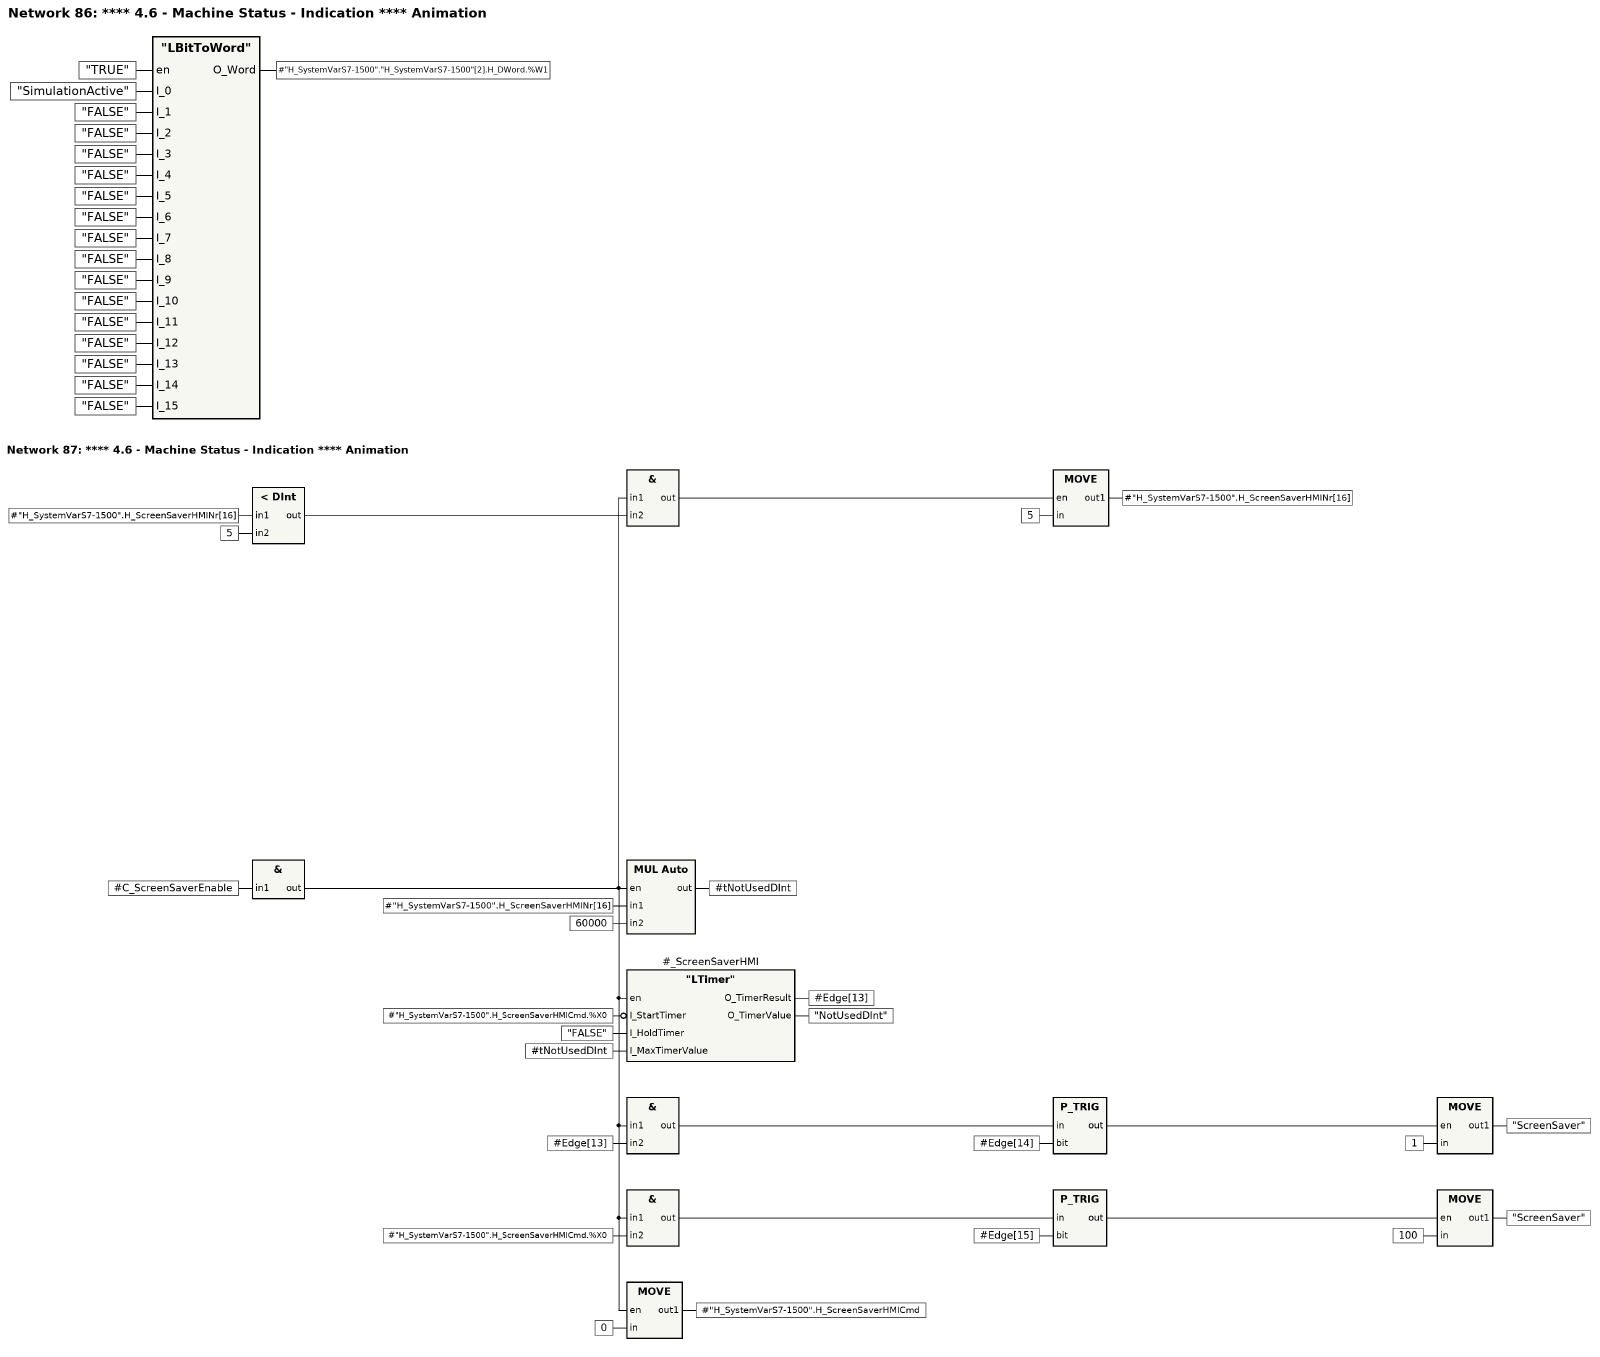
   IF "TRUE" THEN
       "LBitToWord"(I_0 := "SimulationActive",
                    I_1 := "FALSE",
                    I_2 := "FALSE",
                    I_3 := "FALSE",
                    I_4 := "FALSE",
                    I_5 := "FALSE",
                    I_6 := "FALSE",
                    I_7 := "FALSE",
                    I_8 := "FALSE",
                    I_9 := "FALSE",
                    I_10 := "FALSE",
                    I_11 := "FALSE",
                    I_12 := "FALSE",
                    I_13 := "FALSE",
                    I_14 := "FALSE",
                    I_15 := "FALSE",
                    O_Word => #"H_SystemVarS7-1500"."H_SystemVarS7-1500"[2].H_DWord.%W1);
   END_IF;
END_REGION

REGION Network 87: **** 4.6 - Machine Status - Indication **** Animation
   // Animation
   IF #C_ScreenSaverEnable AND (#"H_SystemVarS7-1500".H_ScreenSaverHMINr[16] < 5) THEN
       #"H_SystemVarS7-1500".H_ScreenSaverHMINr[16] := 5;
   END_IF;
   IF #C_ScreenSaverEnable THEN
       #tNotUsedDInt := #"H_SystemVarS7-1500".H_ScreenSaverHMINr[16] * 60000;
       #_ScreenSaverHMI(I_StartTimer := NOT #"H_SystemVarS7-1500".H_ScreenSaverHMICmd.%X0,   // "LTimer"
                        I_HoldTimer := "FALSE",
                        I_MaxTimerValue := #tNotUsedDInt,
                        O_TimerResult => #Edge[13],
                        O_TimerValue => "NotUsedDInt");
   END_IF;
   #_w1 := #C_ScreenSaverEnable AND #Edge[13];
   #_w2 := #_w1 AND NOT #Edge[14];   // rising edge
   #Edge[14] := #_w1;
   IF #_w2 THEN "ScreenSaver" := 1; END_IF;
   #_w3 := #C_ScreenSaverEnable AND #"H_SystemVarS7-1500".H_ScreenSaverHMICmd.%X0;
   #_w4 := #_w3 AND NOT #Edge[15];   // rising edge
   #Edge[15] := #_w3;
   IF #_w4 THEN "ScreenSaver" := 100; END_IF;
   IF #C_ScreenSaverEnable THEN #"H_SystemVarS7-1500".H_ScreenSaverHMICmd := 0; END_IF;
END_REGION

REGION Network 88: **** 4.6 - Machine Status - Indication **** Animation (LED status of the cpu)
   // Animation (LED status of the cpu)
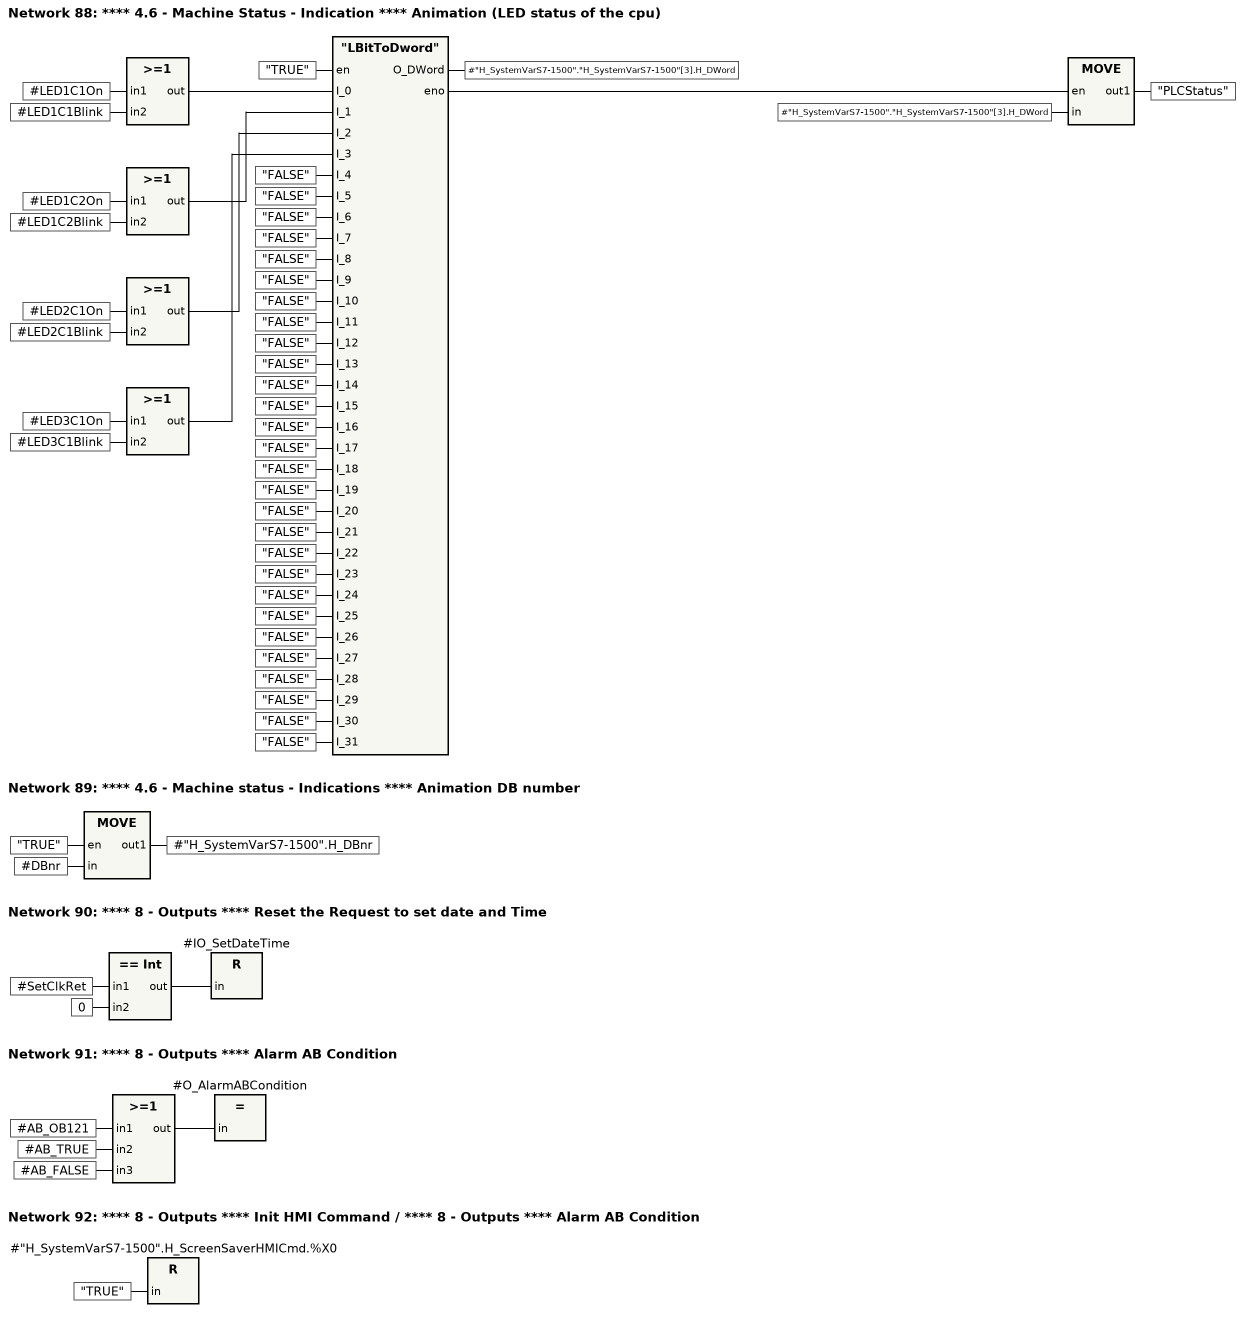
   "LBitToDword"(EN := "TRUE",
                 I_0 := #LED1C1On OR #LED1C1Blink,
                 I_1 := #LED1C2On OR #LED1C2Blink,
                 I_2 := #LED2C1On OR #LED2C1Blink,
                 I_3 := #LED3C1On OR #LED3C1Blink,
                 I_4 := "FALSE",
                 I_5 := "FALSE",
                 I_6 := "FALSE",
                 I_7 := "FALSE",
                 I_8 := "FALSE",
                 I_9 := "FALSE",
                 I_10 := "FALSE",
                 I_11 := "FALSE",
                 I_12 := "FALSE",
                 I_13 := "FALSE",
                 I_14 := "FALSE",
                 I_15 := "FALSE",
                 I_16 := "FALSE",
                 I_17 := "FALSE",
                 I_18 := "FALSE",
                 I_19 := "FALSE",
                 I_20 := "FALSE",
                 I_21 := "FALSE",
                 I_22 := "FALSE",
                 I_23 := "FALSE",
                 I_24 := "FALSE",
                 I_25 := "FALSE",
                 I_26 := "FALSE",
                 I_27 := "FALSE",
                 I_28 := "FALSE",
                 I_29 := "FALSE",
                 I_30 := "FALSE",
                 I_31 := "FALSE",
                 O_DWord => #"H_SystemVarS7-1500"."H_SystemVarS7-1500"[3].H_DWord,
                 ENO => #_w1);
   IF #_w1 THEN "PLCStatus" := #"H_SystemVarS7-1500"."H_SystemVarS7-1500"[3].H_DWord; END_IF;
END_REGION

REGION Network 89: **** 4.6 - Machine status - Indications **** Animation DB number
   // Animation DB number
   IF "TRUE" THEN #"H_SystemVarS7-1500".H_DBnr := #DBnr; END_IF;
END_REGION

REGION Network 90: **** 8 - Outputs **** Reset the Request to set date and Time
   // Reset the Request to set date and Time
   IF #SetClkRet = 0 THEN #IO_SetDateTime := FALSE; END_IF;
END_REGION

REGION Network 91: **** 8 - Outputs **** Alarm AB Condition
   // Alarm AB Condition
   #O_AlarmABCondition := #AB_OB121 OR #AB_TRUE OR #AB_FALSE;
END_REGION

REGION Network 92: **** 8 - Outputs **** Init HMI Command / **** 8 - Outputs **** Alarm AB Condition
   // Init HMI Command / Alarm AB Condition
   IF "TRUE" THEN #"H_SystemVarS7-1500".H_ScreenSaverHMICmd.%X0 := FALSE; END_IF;
END_REGION

REGION Network 93: **** 9 - Alarm Summary **** Alarm A
   // Alarm A
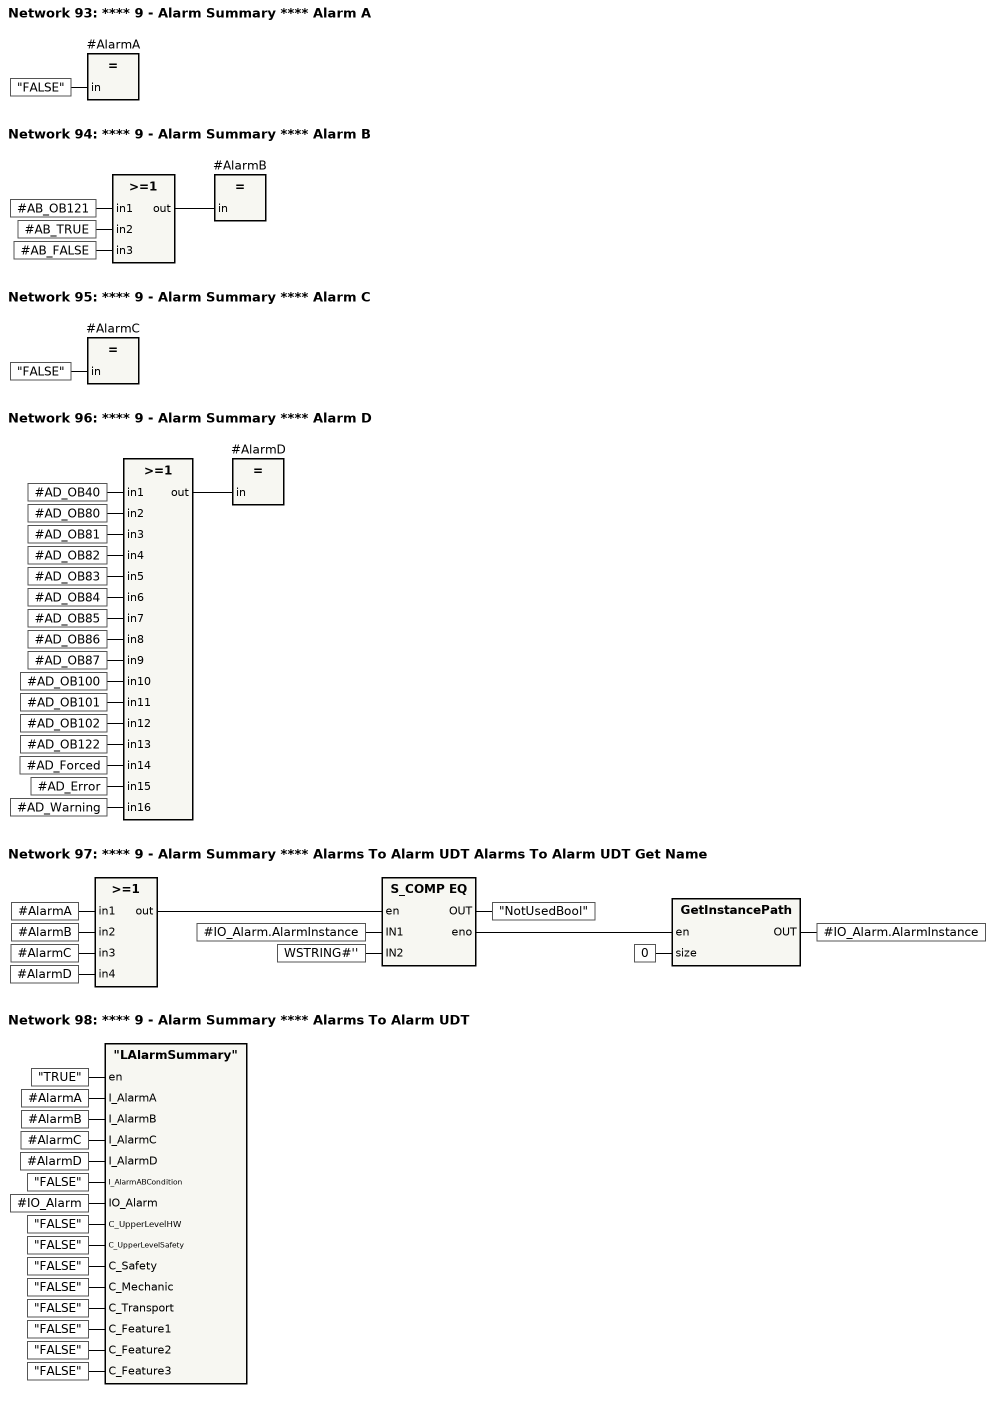
   #AlarmA := "FALSE";
END_REGION

REGION Network 94: **** 9 - Alarm Summary **** Alarm B
   // Alarm B
   #AlarmB := #AB_OB121 OR #AB_TRUE OR #AB_FALSE;
END_REGION

REGION Network 95: **** 9 - Alarm Summary **** Alarm C
   // Alarm C
   #AlarmC := "FALSE";
END_REGION

REGION Network 96: **** 9 - Alarm Summary **** Alarm D
   // Alarm D
   #AlarmD := #AD_OB40 OR #AD_OB80 OR #AD_OB81 OR #AD_OB82 OR #AD_OB83 OR #AD_OB84 OR #AD_OB85 OR #AD_OB86 OR #AD_OB87 OR #AD_OB100 OR #AD_OB101 OR #AD_OB102 OR #AD_OB122 OR #AD_Forced OR #AD_Error OR #AD_Warning;
END_REGION

REGION Network 97: **** 9 - Alarm Summary **** Alarms To Alarm UDT Alarms To Alarm UDT Get Name
   // Alarm / Alarm D
   S_COMP(EN := #AlarmA OR #AlarmB OR #AlarmC OR #AlarmD,
          IN1 := #IO_Alarm.AlarmInstance,
          IN2 := WSTRING#'',
          OUT => "NotUsedBool",
          ENO => #_w1);
   IF #_w1 THEN GetInstancePath(size := 0, OUT => #IO_Alarm.AlarmInstance); END_IF;
END_REGION

REGION Network 98: **** 9 - Alarm Summary **** Alarms To Alarm UDT
   // Alarm / Alarm D
   IF "TRUE" THEN
       "LAlarmSummary"(I_AlarmA := #AlarmA,
                       I_AlarmB := #AlarmB,
                       I_AlarmC := #AlarmC,
                       I_AlarmD := #AlarmD,
                       I_AlarmABCondition := "FALSE",
                       IO_Alarm := #IO_Alarm,
                       C_UpperLevelHW := "FALSE",
                       C_UpperLevelSafety := "FALSE",
                       C_Safety := "FALSE",
                       C_Mechanic := "FALSE",
                       C_Transport := "FALSE",
                       C_Feature1 := "FALSE",
                       C_Feature2 := "FALSE",
                       C_Feature3 := "FALSE");
   END_IF;
END_REGION

REGION Network 99: **** 9.1 - Alarm Output **** Alarm A
   // Alarm A
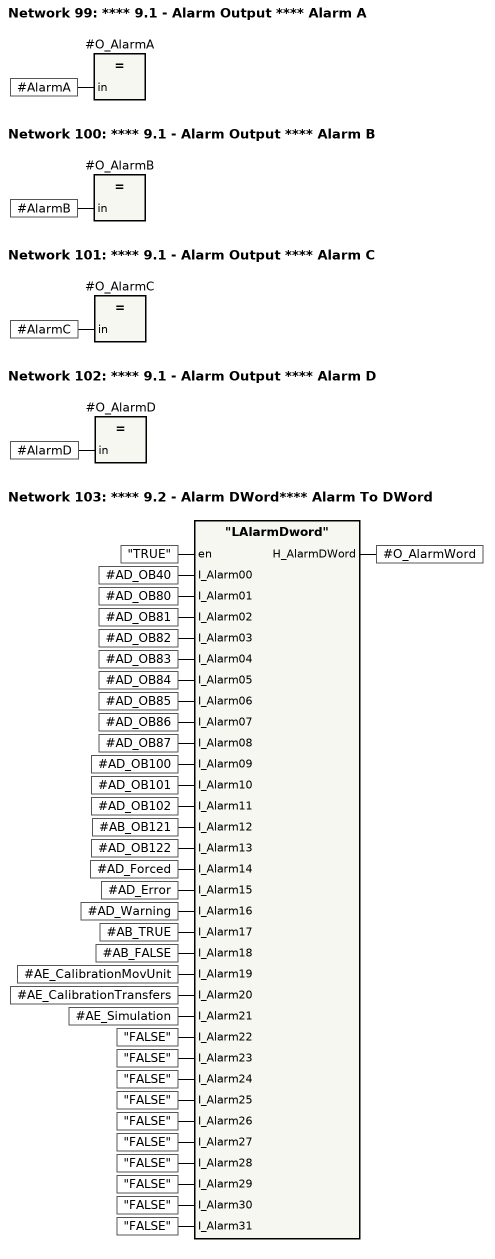
   #O_AlarmA := #AlarmA;
END_REGION

REGION Network 100: **** 9.1 - Alarm Output **** Alarm B
   // Alarm B
   #O_AlarmB := #AlarmB;
END_REGION

REGION Network 101: **** 9.1 - Alarm Output **** Alarm C
   // Alarm C
   #O_AlarmC := #AlarmC;
END_REGION

REGION Network 102: **** 9.1 - Alarm Output **** Alarm D
   // Alarm D
   #O_AlarmD := #AlarmD;
END_REGION

REGION Network 103: **** 9.2 - Alarm DWord**** Alarm To DWord
   // Alarm To Word
   IF "TRUE" THEN
       "LAlarmDword"(I_Alarm00 := #AD_OB40,
                     I_Alarm01 := #AD_OB80,
                     I_Alarm02 := #AD_OB81,
                     I_Alarm03 := #AD_OB82,
                     I_Alarm04 := #AD_OB83,
                     I_Alarm05 := #AD_OB84,
                     I_Alarm06 := #AD_OB85,
                     I_Alarm07 := #AD_OB86,
                     I_Alarm08 := #AD_OB87,
                     I_Alarm09 := #AD_OB100,
                     I_Alarm10 := #AD_OB101,
                     I_Alarm11 := #AD_OB102,
                     I_Alarm12 := #AB_OB121,
                     I_Alarm13 := #AD_OB122,
                     I_Alarm14 := #AD_Forced,
                     I_Alarm15 := #AD_Error,
                     I_Alarm16 := #AD_Warning,
                     I_Alarm17 := #AB_TRUE,
                     I_Alarm18 := #AB_FALSE,
                     I_Alarm19 := #AE_CalibrationMovUnit,
                     I_Alarm20 := #AE_CalibrationTransfers,
                     I_Alarm21 := #AE_Simulation,
                     I_Alarm22 := "FALSE",
                     I_Alarm23 := "FALSE",
                     I_Alarm24 := "FALSE",
                     I_Alarm25 := "FALSE",
                     I_Alarm26 := "FALSE",
                     I_Alarm27 := "FALSE",
                     I_Alarm28 := "FALSE",
                     I_Alarm29 := "FALSE",
                     I_Alarm30 := "FALSE",
                     I_Alarm31 := "FALSE",
                     H_AlarmDWord => #O_AlarmWord);
   END_IF;
END_REGION
END_FUNCTION_BLOCK

FUNCTION_BLOCK "LToggle"   // FB1108, FBD
TITLE = LToggle
{ S7_Optimized_Access := 'TRUE' }
AUTHOR : VCC
FAMILY : Function
NAME : LToggle
VERSION : 0.1
// ================================================================================
// Change the state of the output everytime the input is on
// ================================================================================
// stored: AutoNumber false, IsIECCheckEnabled false, IsRetainMemResEnabled false, MemoryReserve 100, SetENOAutomatically False, UDAEnableTagReadback false
   VAR_INPUT
      I_Input { ExternalAccessible := 'False'; ExternalVisible := 'False'; ExternalWritable := 'False'} : Bool;   // The input
   END_VAR
   VAR_OUTPUT
      O_Output { ExternalAccessible := 'False'; ExternalVisible := 'False'; ExternalWritable := 'False'} : Bool;   // The output
   END_VAR
   VAR RETAIN
      pulseReqOn { ExternalAccessible := 'False'; ExternalVisible := 'False'; ExternalWritable := 'False'} : Bool;   // Pulse request on
      pulseReqOff { ExternalAccessible := 'False'; ExternalVisible := 'False'; ExternalWritable := 'False'} : Bool;   // Pulse request off
      Output { ExternalAccessible := 'False'; ExternalVisible := 'False'; ExternalWritable := 'False'} : Bool;   // Temporary Output
      ReqOutputOff { ExternalAccessible := 'False'; ExternalVisible := 'False'; ExternalWritable := 'False'} : Bool;   // Request output off
      ReqOutputOn { ExternalAccessible := 'False'; ExternalVisible := 'False'; ExternalWritable := 'False'} : Bool;   // Request output on
   END_VAR
   VAR_TEMP   // added for the SCL form of the ladder/FBD networks
      _w1 : Bool;
   END_VAR
BEGIN

REGION Network 1: **** 5.2 - Equations - Flow **** Request on
   // Request on
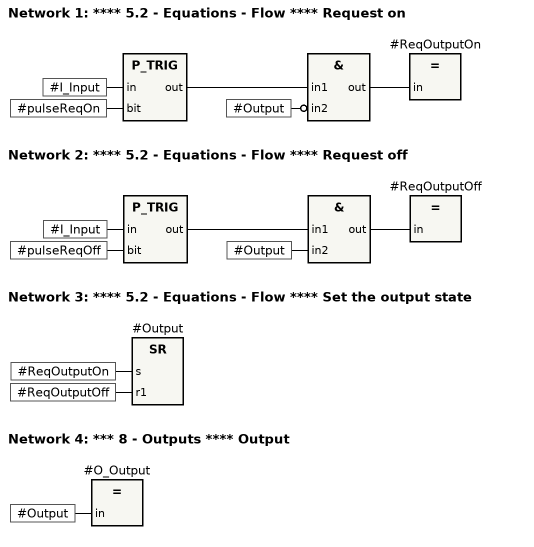
   #_w1 := #I_Input AND NOT #pulseReqOn;   // rising edge
   #pulseReqOn := #I_Input;
   #ReqOutputOn := #_w1 AND NOT #Output;
END_REGION

REGION Network 2: **** 5.2 - Equations - Flow **** Request off
   // Request off
   #_w1 := #I_Input AND NOT #pulseReqOff;   // rising edge
   #pulseReqOff := #I_Input;
   #ReqOutputOff := #_w1 AND #Output;
END_REGION

REGION Network 3: **** 5.2 - Equations - Flow **** Set the output state
   // Set the output state
   IF #ReqOutputOn THEN
       #Output := TRUE;   // SR flip-flop
   END_IF;
   IF #ReqOutputOff THEN #Output := FALSE; END_IF;
END_REGION

REGION Network 4: *** 8 - Outputs **** Output
   // Output
   #O_Output := #Output;
END_REGION
END_FUNCTION_BLOCK

FUNCTION_BLOCK "LTimer"   // FB1009, FBD
TITLE = LTimer
{ S7_Optimized_Access := 'FALSE' }
AUTHOR : VCC
FAMILY : Control
NAME : TimerON
VERSION : 1.0
// ================================================================================
// LTimer is used when a delay is necessary without using a hardware timer.
// The output of the timer will follow the input after a delay time. When the 
// input 
// drops to False, the output will drop immediatly.
// 
// During the activation of timer, hold input can freeze the timer
// * Input Hold = false then normal running of timer
// * Input Hold = true then timer frozen.
// ================================================================================
// stored: AutoNumber false, IsIECCheckEnabled false, SetENOAutomatically False, UDAEnableTagReadback false
   VAR_INPUT
      I_StartTimer { ExternalAccessible := 'False'; ExternalVisible := 'False'; ExternalWritable := 'False'} : Bool;   // Start Timer
      I_HoldTimer { ExternalAccessible := 'False'; ExternalVisible := 'False'; ExternalWritable := 'False'} : Bool;   // Hold timer
      I_MaxTimerValue { ExternalAccessible := 'False'; ExternalVisible := 'False'; ExternalWritable := 'False'} : DInt;   // Maximum Timer Value (1 unit = 1ms and max=7FFFFFFF)
   END_VAR
   VAR_OUTPUT
      O_TimerResult { ExternalAccessible := 'False'; ExternalVisible := 'False'; ExternalWritable := 'False'} : Bool;   // Timer result when time = MaxTime
      O_TimerValue { ExternalAccessible := 'False'; ExternalVisible := 'False'; ExternalWritable := 'False'} : DInt;   // Current timer value
   END_VAR
   VAR DB_SPECIFIC
      PrevCPUSystemTime { ExternalAccessible := 'False'; ExternalVisible := 'False'; ExternalWritable := 'False'} : DInt;   // Last value of the CPU system time register
      DeltaCpuTime { ExternalAccessible := 'False'; ExternalVisible := 'False'; ExternalWritable := 'False'} : DInt;   // Time difference of CPU System Time register compared with last scan
      TempDInt1 { ExternalAccessible := 'False'; ExternalVisible := 'False'; ExternalWritable := 'False'} : DInt;   // Just a temporary Double Integer value
      TimerValue { ExternalAccessible := 'False'; ExternalVisible := 'False'; ExternalWritable := 'False'} : DInt;   // Current timer value
   END_VAR
BEGIN

REGION Network 1: **** 4.4 - Machine Status - Calculated **** Set #TimerValue to zero whenever it a negative.
   // Set #TimerValue to zero whenever it a negative.
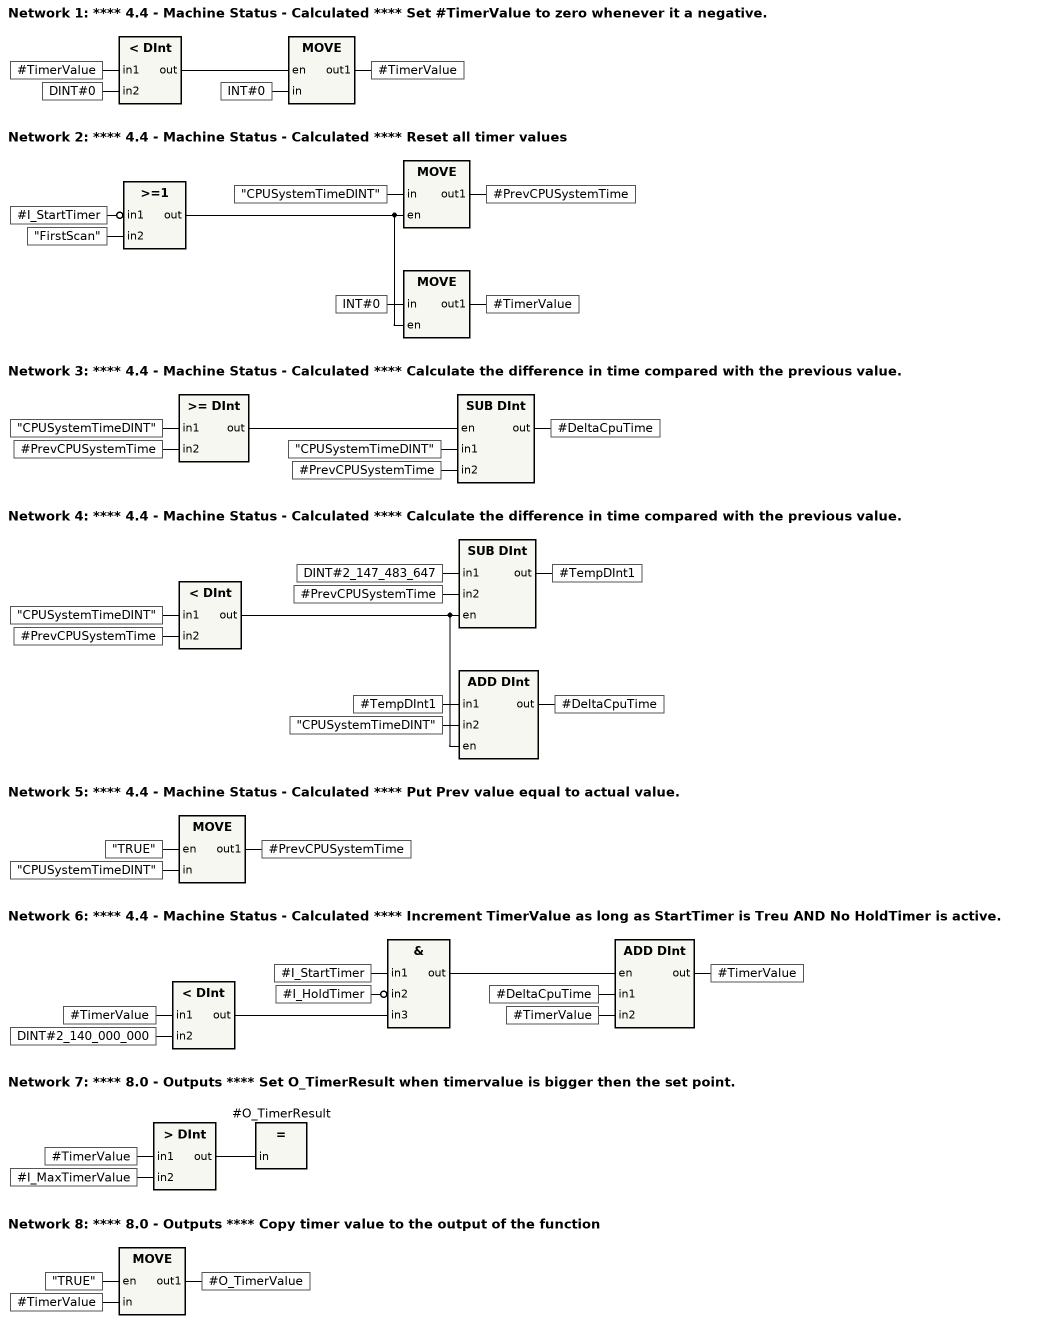
   IF #TimerValue < DINT#0 THEN #TimerValue := INT#0; END_IF;
END_REGION

REGION Network 2: **** 4.4 - Machine Status - Calculated **** Reset all timer values
   // Reset all timer values
   IF NOT #I_StartTimer OR "FirstScan" THEN
       #PrevCPUSystemTime := "CPUSystemTimeDINT";
       #TimerValue := INT#0;
   END_IF;
END_REGION

REGION Network 3: **** 4.4 - Machine Status - Calculated **** Calculate the difference in time compared with the previous value.
   // Calculate the difference in time compared with the previous value.
   IF "CPUSystemTimeDINT" >= #PrevCPUSystemTime THEN
       #DeltaCpuTime := "CPUSystemTimeDINT" - #PrevCPUSystemTime;
   END_IF;
END_REGION

REGION Network 4: **** 4.4 - Machine Status - Calculated **** Calculate the difference in time compared with the previous value.
   // Calculate the difference in time compared with the previous value.
   // If the cpu time has passed 2147483647 then the delta is used first.
   IF "CPUSystemTimeDINT" < #PrevCPUSystemTime THEN
       #TempDInt1 := DINT#2_147_483_647 - #PrevCPUSystemTime;
       #DeltaCpuTime := #TempDInt1 + "CPUSystemTimeDINT";
   END_IF;
END_REGION

REGION Network 5: **** 4.4 - Machine Status - Calculated **** Put Prev value equal to actual value.
   // Put Prev value equal to actual value.
   IF "TRUE" THEN #PrevCPUSystemTime := "CPUSystemTimeDINT"; END_IF;
END_REGION

REGION Network 6: **** 4.4 - Machine Status - Calculated **** Increment TimerValue as long as StartTimer is Treu AND No HoldTimer is active.
   // Increment TimerValue as long as StartTimer is Treu AND No HoldTimer is active.
   // Make sure that there is no override by limiting the increment.
   IF #I_StartTimer AND NOT #I_HoldTimer AND (#TimerValue < DINT#2_140_000_000) THEN
       #TimerValue := #DeltaCpuTime + #TimerValue;
   END_IF;
END_REGION

REGION Network 7: **** 8.0 - Outputs **** Set O_TimerResult when timervalue is bigger then the set point.
   // Set O_TimerResult when timervalue is bigger then the set point.
   #O_TimerResult := #TimerValue > #I_MaxTimerValue;
END_REGION

REGION Network 8: **** 8.0 - Outputs **** Copy timer value to the output of the function
   // Copy timer value to the output of the function
   IF "TRUE" THEN #O_TimerValue := #TimerValue; END_IF;
END_REGION
END_FUNCTION_BLOCK

FUNCTION_BLOCK "LActiveShift"   // FB1800, FBD
TITLE = LActifShift
{ S7_Optimized_Access := 'FALSE' }
AUTHOR : VCC
FAMILY : Supervis
NAME : LActShif
VERSION : 1.0
// ================================================================================
// Module used to give which shift is active with the calendar variable of PLC
// Morning shift: start - stop is defined by HMI
// Evening shift: start - stop is defined by HMI
// Night shift  : start - stop is defined by HMI
// ================================================================================
// stored: AutoNumber false, IsIECCheckEnabled false, SetENOAutomatically False, UDAEnableTagReadback false
   VAR_OUTPUT
      O_MorningShift { ExternalAccessible := 'False'; ExternalVisible := 'False'; ExternalWritable := 'False'} : Bool;   // Morning shift
      O_EveningShift { ExternalAccessible := 'False'; ExternalVisible := 'False'; ExternalWritable := 'False'} : Bool;   // Evening shift
      O_NightShift { ExternalAccessible := 'False'; ExternalVisible := 'False'; ExternalWritable := 'False'} : Bool;   // NightShift
      O_NewShift { ExternalAccessible := 'False'; ExternalVisible := 'False'; ExternalWritable := 'False'} : Bool;   // NewShift / Morning shift
      O_ShiftOverview { ExternalAccessible := 'False'; ExternalVisible := 'False'; ExternalWritable := 'False'} : Struct   // Overview Active Shift
         MorningShift_Day1 { ExternalAccessible := 'False'; ExternalVisible := 'False'; ExternalWritable := 'False'} : Bool;   // Morning Shift of Day 1 (Monday)
         EveningShift_Day1 { ExternalAccessible := 'False'; ExternalVisible := 'False'; ExternalWritable := 'False'} : Bool;   // Evening Shift of Day 1 (Monday)
         NightShift_Day1 { ExternalAccessible := 'False'; ExternalVisible := 'False'; ExternalWritable := 'False'} : Bool;   // Night Shift of Day 1 (Monday-Tuesday)
         MorningShift_Day2 { ExternalAccessible := 'False'; ExternalVisible := 'False'; ExternalWritable := 'False'} : Bool;   // Morning Shift of Day 2 (Tuesday)
         EveningShift_Day2 { ExternalAccessible := 'False'; ExternalVisible := 'False'; ExternalWritable := 'False'} : Bool;   // Evening Shift of Day 2 (Tuesday)
         NightShift_Day2 { ExternalAccessible := 'False'; ExternalVisible := 'False'; ExternalWritable := 'False'} : Bool;   // Night Shift of Day 2 (Tuesday-Wednesday)
         MorningShift_Day3 { ExternalAccessible := 'False'; ExternalVisible := 'False'; ExternalWritable := 'False'} : Bool;   // Morning Shift of Day 3 (Wednesday)
         EveningShift_Day3 { ExternalAccessible := 'False'; ExternalVisible := 'False'; ExternalWritable := 'False'} : Bool;   // Evening Shift of Day 3 (Wednesday)
         NightShift_Day3 { ExternalAccessible := 'False'; ExternalVisible := 'False'; ExternalWritable := 'False'} : Bool;   // night Shift of Day 3 (Wednesday-Thursday)
         MorningShift_Day4 { ExternalAccessible := 'False'; ExternalVisible := 'False'; ExternalWritable := 'False'} : Bool;   // Morning Shift of Day 4 (Thursday)
         EveningShift_Day4 { ExternalAccessible := 'False'; ExternalVisible := 'False'; ExternalWritable := 'False'} : Bool;   // Evening Shift of Day 4 (Thursday)
         NightShift_Day4 { ExternalAccessible := 'False'; ExternalVisible := 'False'; ExternalWritable := 'False'} : Bool;   // Night Shift of Day 4 (Thursday-Friday)
         MorningShift_Day5 { ExternalAccessible := 'False'; ExternalVisible := 'False'; ExternalWritable := 'False'} : Bool;   // Morning Shift of Day 5 (Friday)
         EveningShift_Day5 { ExternalAccessible := 'False'; ExternalVisible := 'False'; ExternalWritable := 'False'} : Bool;   // Evening Shift of Day 5 (Friday)
         NightShift_Day5 { ExternalAccessible := 'False'; ExternalVisible := 'False'; ExternalWritable := 'False'} : Bool;   // Night Shift of Day 5 (Friday-Saturday)
         MorningShift_Day6 { ExternalAccessible := 'False'; ExternalVisible := 'False'; ExternalWritable := 'False'} : Bool;   // Morning Shift of Day 6 (Saturday)
         EveningShift_Day6 { ExternalAccessible := 'False'; ExternalVisible := 'False'; ExternalWritable := 'False'} : Bool;   // Evening Shift of Day 6 (Saturday)
         NightShift_Day6 { ExternalAccessible := 'False'; ExternalVisible := 'False'; ExternalWritable := 'False'} : Bool;   // Night Shift of Day 6 (Saturday-Sunday)
         MorningShift_Day7 { ExternalAccessible := 'False'; ExternalVisible := 'False'; ExternalWritable := 'False'} : Bool;   // Morning Shift of Day 7 (Sunday)
         EveningShift_Day7 { ExternalAccessible := 'False'; ExternalVisible := 'False'; ExternalWritable := 'False'} : Bool;   // Evening Shift of Day 7 (Sunday)
         NightShift_Day7 { ExternalAccessible := 'False'; ExternalVisible := 'False'; ExternalWritable := 'False'} : Bool;   // night Shift of Day 7 (Sunday-Monday)
      END_STRUCT;
      H_IAnim { ExternalAccessible := 'False'; ExternalVisible := 'False'; ExternalWritable := 'False'} : Word;   // HMI Animation of the icon
   END_VAR
   VAR DB_SPECIFIC
      H_In : Struct   // HMI
         StartMorningDay1 : Real := 5.15;   // Start time of morning shift - Day 1
         StartEveningDay1 : Real := 13.15;   // Start time of evening shift - Day 1
         StartNightDay1 : Real := 21.15;   // Start time of night shift - Day 1
         StartMorningDay2 : Real := 5.15;   // Start time of morning shift - Day 2
         StartEveningDay2 : Real := 13.15;   // Start time of evening shift - Day 2
         StartNightDay2 : Real := 21.15;   // Start time of night shift - Day 2
         StartMorningDay3 : Real := 5.15;   // Start time of morning shift - Day 3
         StartEveningDay3 : Real := 13.15;   // Start time of evening shift - Day 3
         StartNightDay3 : Real := 21.15;   // Start time of night shift - Day 3
         StartMorningDay4 : Real := 5.15;   // Start time of morning shift - Day 4
         StartEveningDay4 : Real := 13.15;   // Start time of evening shift - Day 4
         StartNightDay4 : Real := 21.15;   // Start time of night shift - Day 4
         StartMorningDay5 : Real := 5.15;   // Start time of morning shift - Day 5
         StartEveningDay5 : Real := 12.25;   // Start time of evening shift - Day 5
         StartNightDay5 : Real := 19.35;   // Start time of night shift - Day 5
         StartMorningDay6 : Real := 5.15;   // Start time of morning shift - Day 6
         StartEveningDay6 : Real := 13.15;   // Start time of evening shift - Day 6
         StartNightDay6 : Real := 21.15;   // Start time of night shift - Day 6
         StartMorningDay7 : Real := 5.15;   // Start time of morning shift - Day 7
         StartEveningDay7 : Real := 13.15;   // Start time of evening shift - Day 7
         StartNightDay7 : Real := 21.15;   // Start time of night shift - Day 7
      END_STRUCT;
      H_Out : Struct   // HMI
         Anim : Word;   // HMI Animation of the object
         DBnr : Int;   // HMI Animation DB number
      END_STRUCT;
      MorningShift_Day1 { ExternalAccessible := 'False'; ExternalVisible := 'False'; ExternalWritable := 'False'} : Bool;   // Morning Shift of Day 1 (Monday)
      EveningShift_Day1 { ExternalAccessible := 'False'; ExternalVisible := 'False'; ExternalWritable := 'False'} : Bool;   // Evening Shift of Day 1 (Monday)
      NightShift_Day1 { ExternalAccessible := 'False'; ExternalVisible := 'False'; ExternalWritable := 'False'} : Bool;   // Night Shift of Day 1 (Monday-Tuesday)
      MorningShift_Day2 { ExternalAccessible := 'False'; ExternalVisible := 'False'; ExternalWritable := 'False'} : Bool;   // Morning Shift of Day 2 (Tuesday)
      EveningShift_Day2 { ExternalAccessible := 'False'; ExternalVisible := 'False'; ExternalWritable := 'False'} : Bool;   // Evening Shift of Day 2 (Tuesday)
      NightShift_Day2 { ExternalAccessible := 'False'; ExternalVisible := 'False'; ExternalWritable := 'False'} : Bool;   // Night Shift of Day 2 (Tuesday-Wednesday)
      MorningShift_Day3 { ExternalAccessible := 'False'; ExternalVisible := 'False'; ExternalWritable := 'False'} : Bool;   // Morning Shift of Day 3 (Wednesday)
      EveningShift_Day3 { ExternalAccessible := 'False'; ExternalVisible := 'False'; ExternalWritable := 'False'} : Bool;   // Evening Shift of Day 3 (Wednesday)
      NightShift_Day3 { ExternalAccessible := 'False'; ExternalVisible := 'False'; ExternalWritable := 'False'} : Bool;   // night Shift of Day 3 (Wednesday-Thursday)
      MorningShift_Day4 { ExternalAccessible := 'False'; ExternalVisible := 'False'; ExternalWritable := 'False'} : Bool;   // Morning Shift of Day 4 (Thursday)
      EveningShift_Day4 { ExternalAccessible := 'False'; ExternalVisible := 'False'; ExternalWritable := 'False'} : Bool;   // Evening Shift of Day 4 (Thursday)
      NightShift_Day4 { ExternalAccessible := 'False'; ExternalVisible := 'False'; ExternalWritable := 'False'} : Bool;   // Night Shift of Day 4 (Thursday-Friday)
      MorningShift_Day5 { ExternalAccessible := 'False'; ExternalVisible := 'False'; ExternalWritable := 'False'} : Bool;   // Morning Shift of Day 5 (Friday)
      EveningShift_Day5 { ExternalAccessible := 'False'; ExternalVisible := 'False'; ExternalWritable := 'False'} : Bool;   // Evening Shift of Day 5 (Friday)
      NightShift_Day5 { ExternalAccessible := 'False'; ExternalVisible := 'False'; ExternalWritable := 'False'} : Bool;   // Night Shift of Day 5 (Friday-Saturday)
      MorningShift_Day6 { ExternalAccessible := 'False'; ExternalVisible := 'False'; ExternalWritable := 'False'} : Bool;   // Morning Shift of Day 6 (Saturday)
      EveningShift_Day6 { ExternalAccessible := 'False'; ExternalVisible := 'False'; ExternalWritable := 'False'} : Bool;   // Evening Shift of Day 6 (Saturday)
      NightShift_Day6 { ExternalAccessible := 'False'; ExternalVisible := 'False'; ExternalWritable := 'False'} : Bool;   // Night Shift of Day 6 (Saturday-Sunday)
      MorningShift_Day7 { ExternalAccessible := 'False'; ExternalVisible := 'False'; ExternalWritable := 'False'} : Bool;   // Morning Shift of Day 7 (Sunday)
      EveningShift_Day7 { ExternalAccessible := 'False'; ExternalVisible := 'False'; ExternalWritable := 'False'} : Bool;   // Evening Shift of Day 7 (Sunday)
      NightShift_Day7 { ExternalAccessible := 'False'; ExternalVisible := 'False'; ExternalWritable := 'False'} : Bool;   // night Shift of Day 7 (Sunday-Monday)
      MorningShift { ExternalAccessible := 'False'; ExternalVisible := 'False'; ExternalWritable := 'False'} : Bool;   // Morning shift
      EveningShift { ExternalAccessible := 'False'; ExternalVisible := 'False'; ExternalWritable := 'False'} : Bool;   // Evening shift
      NightShift { ExternalAccessible := 'False'; ExternalVisible := 'False'; ExternalWritable := 'False'} : Bool;   // NightShift
      NewShift { ExternalAccessible := 'False'; ExternalVisible := 'False'; ExternalWritable := 'False'} : Bool;   // NewShift / Morning shift
      NewMorningShiftTrig { ExternalAccessible := 'False'; ExternalVisible := 'False'; ExternalWritable := 'False'} : Bool;   // Trigger for New Morning shift / Morning shift
      NewEveningShiftTrig { ExternalAccessible := 'False'; ExternalVisible := 'False'; ExternalWritable := 'False'} : Bool;   // Trigger for New Evening shift / Evening shift
      NewNightShiftTrig { ExternalAccessible := 'False'; ExternalVisible := 'False'; ExternalWritable := 'False'} : Bool;   // Trigger for New NightShift / NightShift
      Day1 { ExternalAccessible := 'False'; ExternalVisible := 'False'; ExternalWritable := 'False'} : Bool;   // Day 1 = Monday
      Day2 { ExternalAccessible := 'False'; ExternalVisible := 'False'; ExternalWritable := 'False'} : Bool;   // Day 2 = Tuesday
      Day3 { ExternalAccessible := 'False'; ExternalVisible := 'False'; ExternalWritable := 'False'} : Bool;   // Day 3 = Wednesday
      Day4 { ExternalAccessible := 'False'; ExternalVisible := 'False'; ExternalWritable := 'False'} : Bool;   // Day 4 = Thursday
      Day5 { ExternalAccessible := 'False'; ExternalVisible := 'False'; ExternalWritable := 'False'} : Bool;   // Day 5 = Friday
      Day6 { ExternalAccessible := 'False'; ExternalVisible := 'False'; ExternalWritable := 'False'} : Bool;   // Day 6 = Saturday
      Day7 { ExternalAccessible := 'False'; ExternalVisible := 'False'; ExternalWritable := 'False'} : Bool;   // Day 7 = Sunday
      Day1_Int_Morning { ExternalAccessible := 'False'; ExternalVisible := 'False'; ExternalWritable := 'False'} : Int := 515;   // Start integer of morning shift - Day 1
      Day1_Int_Evening { ExternalAccessible := 'False'; ExternalVisible := 'False'; ExternalWritable := 'False'} : Int := 1315;   // Start integer of evening shift - Day 1
      Day1_Int_Night { ExternalAccessible := 'False'; ExternalVisible := 'False'; ExternalWritable := 'False'} : Int := 2115;   // Start integer of night shift - Day 1
      Day2_Int_Morning { ExternalAccessible := 'False'; ExternalVisible := 'False'; ExternalWritable := 'False'} : Int := 515;   // Start integer of morning shift - Day 2
      Day2_Int_Evening { ExternalAccessible := 'False'; ExternalVisible := 'False'; ExternalWritable := 'False'} : Int := 1315;   // Start integer of evening shift - Day 2
      Day2_Int_Night { ExternalAccessible := 'False'; ExternalVisible := 'False'; ExternalWritable := 'False'} : Int := 2115;   // Start integer of night shift - Day 2
      Day3_Int_Morning { ExternalAccessible := 'False'; ExternalVisible := 'False'; ExternalWritable := 'False'} : Int := 515;   // Start integer of morning shift - Day 3
      Day3_Int_Evening { ExternalAccessible := 'False'; ExternalVisible := 'False'; ExternalWritable := 'False'} : Int := 1315;   // Start integer of evening shift - Day 3
      Day3_Int_Night { ExternalAccessible := 'False'; ExternalVisible := 'False'; ExternalWritable := 'False'} : Int := 2115;   // Start integer of night shift - Day 3
      Day4_Int_Morning { ExternalAccessible := 'False'; ExternalVisible := 'False'; ExternalWritable := 'False'} : Int := 515;   // Start integer of morning shift - Day 4
      Day4_Int_Evening { ExternalAccessible := 'False'; ExternalVisible := 'False'; ExternalWritable := 'False'} : Int := 1315;   // Start integer of evening shift - Day 4
      Day4_Int_Night { ExternalAccessible := 'False'; ExternalVisible := 'False'; ExternalWritable := 'False'} : Int := 2115;   // Start integer of night shift - Day 4
      Day5_Int_Morning { ExternalAccessible := 'False'; ExternalVisible := 'False'; ExternalWritable := 'False'} : Int := 515;   // Start integer of morning shift - Day 5
      Day5_Int_Evening { ExternalAccessible := 'False'; ExternalVisible := 'False'; ExternalWritable := 'False'} : Int := 1225;   // Start integer of evening shift - Day 5
      Day5_Int_Night { ExternalAccessible := 'False'; ExternalVisible := 'False'; ExternalWritable := 'False'} : Int := 1935;   // Start integer of night shift - Day 5
      Day6_Int_Morning { ExternalAccessible := 'False'; ExternalVisible := 'False'; ExternalWritable := 'False'} : Int := 515;   // Start integer of morning shift - Day 6
      Day6_Int_Evening { ExternalAccessible := 'False'; ExternalVisible := 'False'; ExternalWritable := 'False'} : Int := 1315;   // Start integer of evening shift - Day 6
      Day6_Int_Night { ExternalAccessible := 'False'; ExternalVisible := 'False'; ExternalWritable := 'False'} : Int := 2115;   // Start integer of night shift - Day 6
      Day7_Int_Morning { ExternalAccessible := 'False'; ExternalVisible := 'False'; ExternalWritable := 'False'} : Int := 515;   // Start integer of morning shift - Day 7
      Day7_Int_Evening { ExternalAccessible := 'False'; ExternalVisible := 'False'; ExternalWritable := 'False'} : Int := 1315;   // Start integer of evening shift - Day 7
      Day7_Int_Night { ExternalAccessible := 'False'; ExternalVisible := 'False'; ExternalWritable := 'False'} : Int := 2115;   // Start integer of night shift - Day 7
      DBnr { ExternalAccessible := 'False'; ExternalVisible := 'False'; ExternalWritable := 'False'} : Int;   // HMI DB number
   END_VAR
   VAR_TEMP
      Temp1 : Real;
      Temp2 : Int;
   END_VAR
   VAR_TEMP   // added for the SCL form of the ladder/FBD networks
      _w1 : Bool;
      _w2 : Bool;
      _w3 : Bool;
   END_VAR
BEGIN

NETWORK
TITLE = **** 1 - Inputs **** DB number
// DB number
      L     DINO;
      T     #DBnr;

NETWORK
TITLE = **** 4.4 - Machine status - Calculated **** Copy time from HMI to integer
// Copy time from HMI to integer
//********************** Time day 1 *****************************
      L     #H_In.StartMorningDay1;  // Load Start time of morning shift - Day 1
      L     100.0;  // * 100
      *R;  // *
      RND;  // Conversion real to integer
      T     #Day1_Int_Morning;  // Load start time of morning shift = Day 1

      L     #H_In.StartEveningDay1;  // Load Start time of evening shift - Day 1
      L     100.0;  // * 100
      *R;  // *
      RND;  // Conversion real to integer
      T     #Day1_Int_Evening;  // Load start time of evening shift = Day 1

      L     #H_In.StartNightDay1;  // Load Start time of night shift - Day 1
      L     100.0;  // * 100
      *R;  // *
      RND;  // Conversion real to integer
      T     #Day1_Int_Night;  // Load start time of night shift = Day 1


//********************** Time day 2 *****************************
      L     #H_In.StartMorningDay2;  // Load Start time of morning shift - Day 2
      L     100.0;  // * 100
      *R;  // *
      RND;  // Conversion real to integer
      T     #Day2_Int_Morning;  // Load start time of morning shift = Day 2

      L     #H_In.StartEveningDay2;  // Load Start time of evening shift - Day 2
      L     100.0;  // * 100
      *R;  // *
      RND;  // Conversion real to integer
      T     #Day2_Int_Evening;  // Load start time of evening shift = Day 2

      L     #H_In.StartNightDay2;  // Load Start time of night shift - Day 2
      L     100.0;  // * 100
      *R;  // *
      RND;  // Conversion real to integer
      T     #Day2_Int_Night;  // Load start time of night shift = Day 2

//********************** Time day 3 *****************************
      L     #H_In.StartMorningDay3;  // Load Start time of morning shift - Day 3
      L     100.0;  // * 100
      *R;  // *
      RND;  // Conversion real to integer
      T     #Day3_Int_Morning;  // Load start time of morning shift = Day 3

      L     #H_In.StartEveningDay3;  // Load Start time of evening shift - Day 3
      L     100.0;  // * 100
      *R;  // *
      RND;  // Conversion real to integer
      T     #Day3_Int_Evening;  // Load start time of evening shift = Day 3

      L     #H_In.StartNightDay3;  // Load Start time of night shift - Day 3
      L     100.0;  // * 100
      *R;  // *
      RND;  // Conversion real to integer
      T     #Day3_Int_Night;  // Load start time of night shift = Day 3

//********************** Time day 4 *****************************
      L     #H_In.StartMorningDay4;  // Load Start time of morning shift - Day 4
      L     100.0;  // * 100
      *R;  // *
      RND;  // Conversion real to integer
      T     #Day4_Int_Morning;  // Load start time of morning shift = Day 4

      L     #H_In.StartEveningDay4;  // Load Start time of evening shift - Day 4
      L     100.0;  // * 100
      *R;  // *
      RND;  // Conversion real to integer
      T     #Day4_Int_Evening;  // Load start time of evening shift = Day 4

      L     #H_In.StartNightDay4;  // Load Start time of night shift - Day 4
      L     100.0;  // * 100
      *R;  // *
      RND;  // Conversion real to integer
      T     #Day4_Int_Night;  // Load start time of night shift = Day 4

//********************** Time day 5 *****************************
      L     #H_In.StartMorningDay5;  // Load Start time of morning shift - Day 5
      L     100.0;  // * 100
      *R;  // *
      RND;  // Conversion real to integer
      T     #Day5_Int_Morning;  // Load start time of morning shift = Day 5

      L     #H_In.StartEveningDay5;  // Load Start time of evening shift - Day 5
      L     100.0;  // * 100
      *R;  // *
      RND;  // Conversion real to integer
      T     #Day5_Int_Evening;  // Load start time of evening shift = Day 5

      L     #H_In.StartNightDay5;  // Load Start time of night shift - Day 5
      L     100.0;  // * 100
      *R;  // *
      RND;  // Conversion real to integer
      T     #Day5_Int_Night;  // Load start time of night shift = Day 5

//********************** Time day 6 *****************************
      L     #H_In.StartMorningDay6;  // Load Start time of morning shift - Day 6
      L     100.0;  // * 100
      *R;  // *
      RND;  // Conversion real to integer
      T     #Day6_Int_Morning;  // Load start time of morning shift = Day 6

      L     #H_In.StartEveningDay6;  // Load Start time of evening shift - Day 6
      L     100.0;  // * 100
      *R;  // *
      RND;  // Conversion real to integer
      T     #Day6_Int_Evening;  // Load start time of evening shift = Day 6

      L     #H_In.StartNightDay6;  // Load Start time of night shift - Day 6
      L     100.0;  // * 100
      *R;  // *
      RND;  // Conversion real to integer
      T     #Day6_Int_Night;  // Load start time of night shift = Day 6

//********************** Time day 7 *****************************
      L     #H_In.StartMorningDay7;  // Load Start time of morning shift - Day 7
      L     100.0;  // * 100
      *R;  // *
      RND;  // Conversion real to integer
      T     #Day7_Int_Morning;  // Load start time of morning shift = Day 7

      L     #H_In.StartEveningDay7;  // Load Start time of evening shift - Day 7
      L     100.0;  // * 100
      *R;  // *
      RND;  // Conversion real to integer
      T     #Day7_Int_Evening;  // Load start time of evening shift = Day 7

      L     #H_In.StartNightDay7;  // Load Start time of night shift - Day 7
      L     100.0;  // * 100
      *R;  // *
      RND;  // Conversion real to integer
      T     #Day7_Int_Night;  // Load start time of night shift = Day 7

REGION Network 3: **** 4.4 - Machine status - Calculated **** Morning Shift of Day 1
   // Morning Shift of Day 1
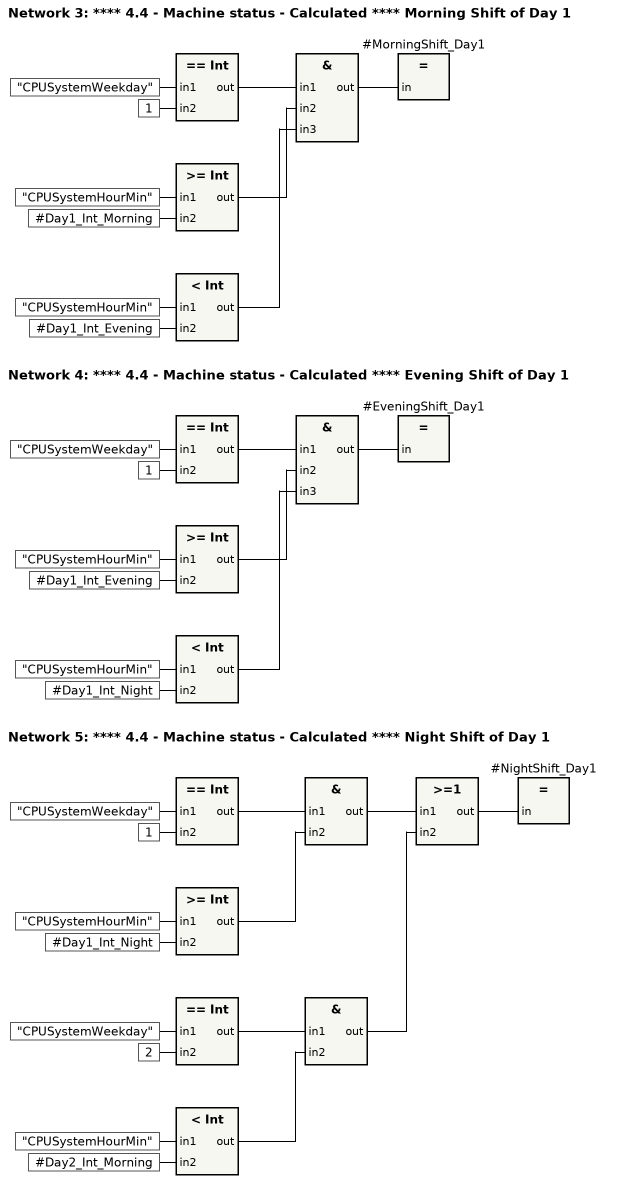
   #MorningShift_Day1 := ("CPUSystemWeekday" = 1) AND ("CPUSystemHourMin" >= #Day1_Int_Morning) AND ("CPUSystemHourMin" < #Day1_Int_Evening);
END_REGION

REGION Network 4: **** 4.4 - Machine status - Calculated **** Evening Shift of Day 1
   // Evening Shift of Day 1
   #EveningShift_Day1 := ("CPUSystemWeekday" = 1) AND ("CPUSystemHourMin" >= #Day1_Int_Evening) AND ("CPUSystemHourMin" < #Day1_Int_Night);
END_REGION

REGION Network 5: **** 4.4 - Machine status - Calculated **** Night Shift of Day 1
   // Night Shift of Day 1
   #NightShift_Day1 := (("CPUSystemWeekday" = 1) AND ("CPUSystemHourMin" >= #Day1_Int_Night)) OR (("CPUSystemWeekday" = 2) AND ("CPUSystemHourMin" < #Day2_Int_Morning));
END_REGION

REGION Network 6: **** 4.4 - Machine status - Calculated **** Morning Shift of Day 2
   // Morning Shift of Day 2
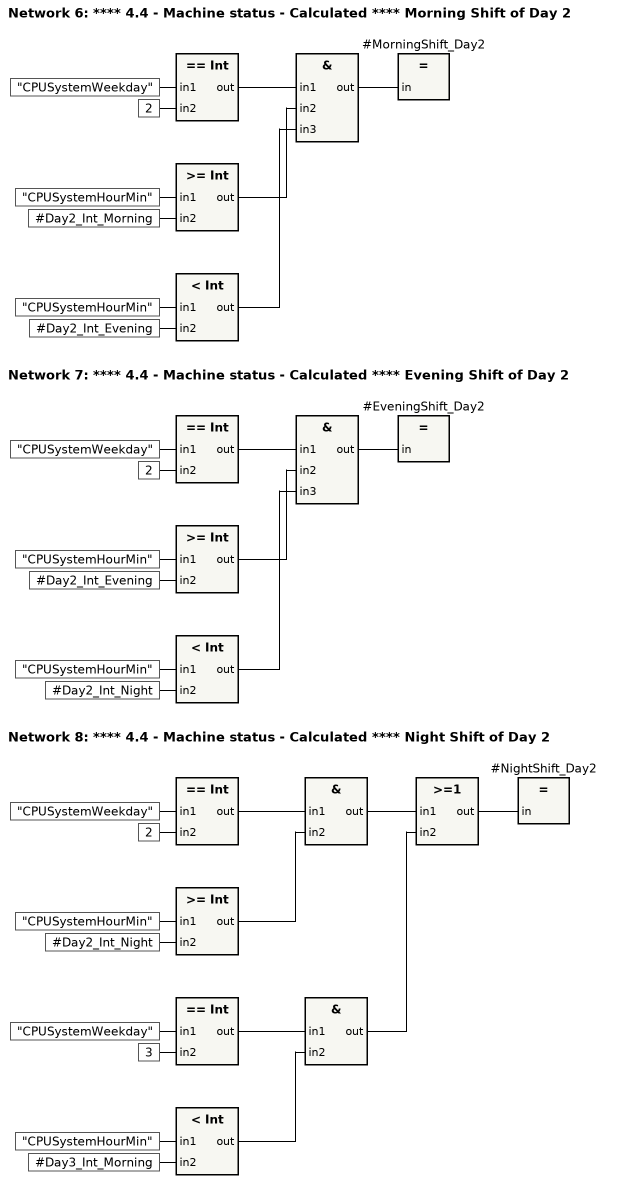
   #MorningShift_Day2 := ("CPUSystemWeekday" = 2) AND ("CPUSystemHourMin" >= #Day2_Int_Morning) AND ("CPUSystemHourMin" < #Day2_Int_Evening);
END_REGION

REGION Network 7: **** 4.4 - Machine status - Calculated **** Evening Shift of Day 2
   // Evening Shift of Day 2
   #EveningShift_Day2 := ("CPUSystemWeekday" = 2) AND ("CPUSystemHourMin" >= #Day2_Int_Evening) AND ("CPUSystemHourMin" < #Day2_Int_Night);
END_REGION

REGION Network 8: **** 4.4 - Machine status - Calculated **** Night Shift of Day 2
   // Night Shift of Day 2
   #NightShift_Day2 := (("CPUSystemWeekday" = 2) AND ("CPUSystemHourMin" >= #Day2_Int_Night)) OR (("CPUSystemWeekday" = 3) AND ("CPUSystemHourMin" < #Day3_Int_Morning));
END_REGION

REGION Network 9: **** 4.4 - Machine status - Calculated **** Morning Shift of Day 3
   // Morning Shift of Day 3
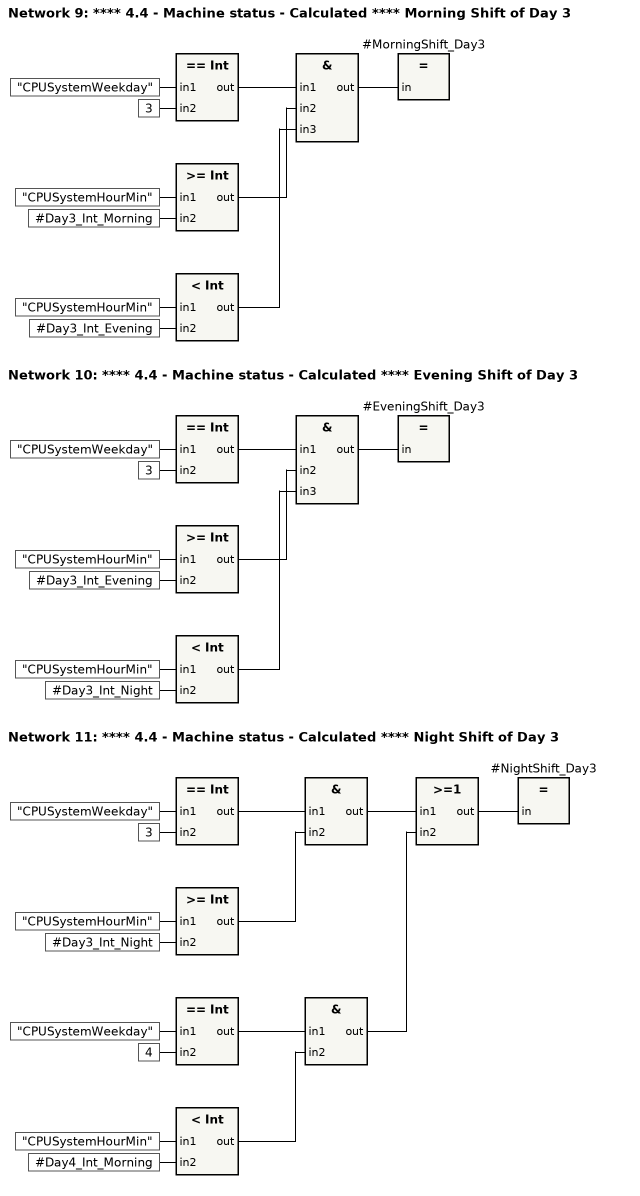
   #MorningShift_Day3 := ("CPUSystemWeekday" = 3) AND ("CPUSystemHourMin" >= #Day3_Int_Morning) AND ("CPUSystemHourMin" < #Day3_Int_Evening);
END_REGION

REGION Network 10: **** 4.4 - Machine status - Calculated **** Evening Shift of Day 3
   // Evening Shift of Day 3
   #EveningShift_Day3 := ("CPUSystemWeekday" = 3) AND ("CPUSystemHourMin" >= #Day3_Int_Evening) AND ("CPUSystemHourMin" < #Day3_Int_Night);
END_REGION

REGION Network 11: **** 4.4 - Machine status - Calculated **** Night Shift of Day 3
   // Night Shift of Day 3
   #NightShift_Day3 := (("CPUSystemWeekday" = 3) AND ("CPUSystemHourMin" >= #Day3_Int_Night)) OR (("CPUSystemWeekday" = 4) AND ("CPUSystemHourMin" < #Day4_Int_Morning));
END_REGION

REGION Network 12: **** 4.4 - Machine status - Calculated **** Morning Shift of Day 4
   // Morning Shift of Day 4
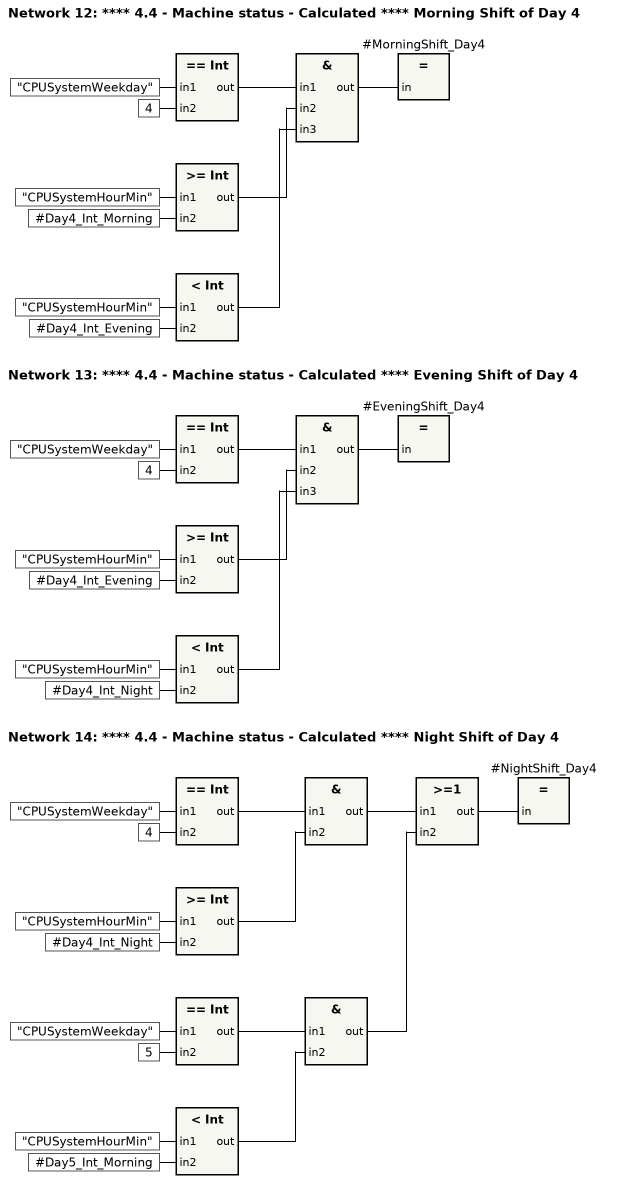
   #MorningShift_Day4 := ("CPUSystemWeekday" = 4) AND ("CPUSystemHourMin" >= #Day4_Int_Morning) AND ("CPUSystemHourMin" < #Day4_Int_Evening);
END_REGION

REGION Network 13: **** 4.4 - Machine status - Calculated **** Evening Shift of Day 4
   // Evening Shift of Day 4
   #EveningShift_Day4 := ("CPUSystemWeekday" = 4) AND ("CPUSystemHourMin" >= #Day4_Int_Evening) AND ("CPUSystemHourMin" < #Day4_Int_Night);
END_REGION

REGION Network 14: **** 4.4 - Machine status - Calculated **** Night Shift of Day 4
   // Night Shift of Day 4
   #NightShift_Day4 := (("CPUSystemWeekday" = 4) AND ("CPUSystemHourMin" >= #Day4_Int_Night)) OR (("CPUSystemWeekday" = 5) AND ("CPUSystemHourMin" < #Day5_Int_Morning));
END_REGION

REGION Network 15: **** 4.4 - Machine status - Calculated **** Morning Shift of Day 5
   // Morning Shift of Day 5
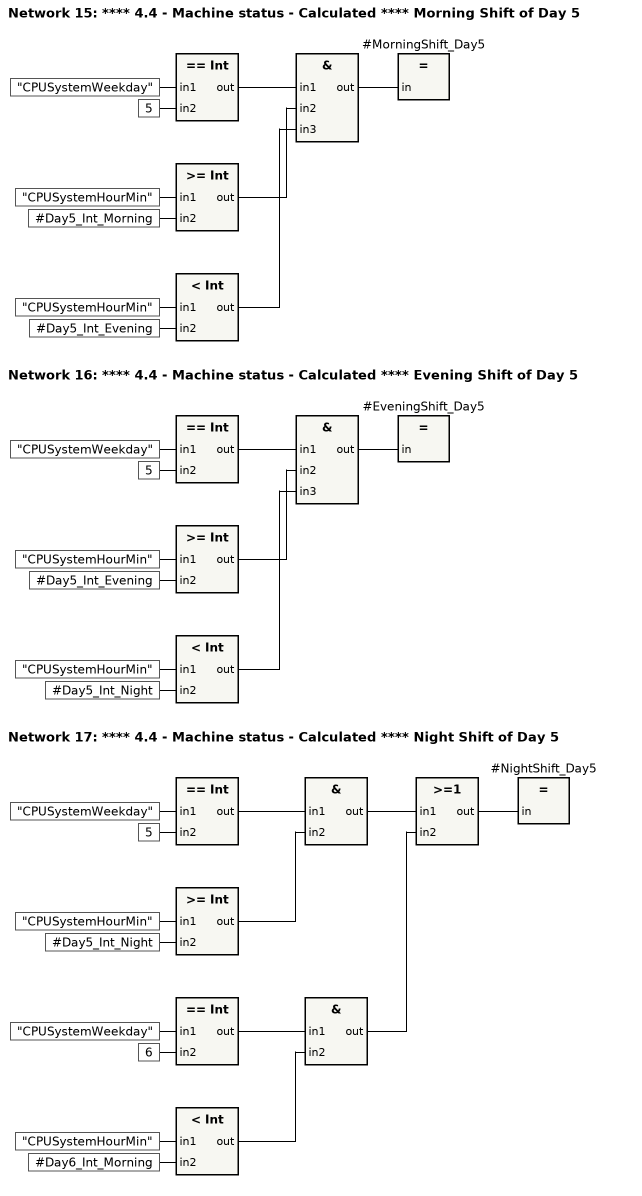
   #MorningShift_Day5 := ("CPUSystemWeekday" = 5) AND ("CPUSystemHourMin" >= #Day5_Int_Morning) AND ("CPUSystemHourMin" < #Day5_Int_Evening);
END_REGION

REGION Network 16: **** 4.4 - Machine status - Calculated **** Evening Shift of Day 5
   // Evening Shift of Day 5
   #EveningShift_Day5 := ("CPUSystemWeekday" = 5) AND ("CPUSystemHourMin" >= #Day5_Int_Evening) AND ("CPUSystemHourMin" < #Day5_Int_Night);
END_REGION

REGION Network 17: **** 4.4 - Machine status - Calculated **** Night Shift of Day 5
   // Night Shift of Day 5
   #NightShift_Day5 := (("CPUSystemWeekday" = 5) AND ("CPUSystemHourMin" >= #Day5_Int_Night)) OR (("CPUSystemWeekday" = 6) AND ("CPUSystemHourMin" < #Day6_Int_Morning));
END_REGION

REGION Network 18: **** 4.4 - Machine status - Calculated **** Morning Shift of Day 6
   // Morning Shift of Day 6
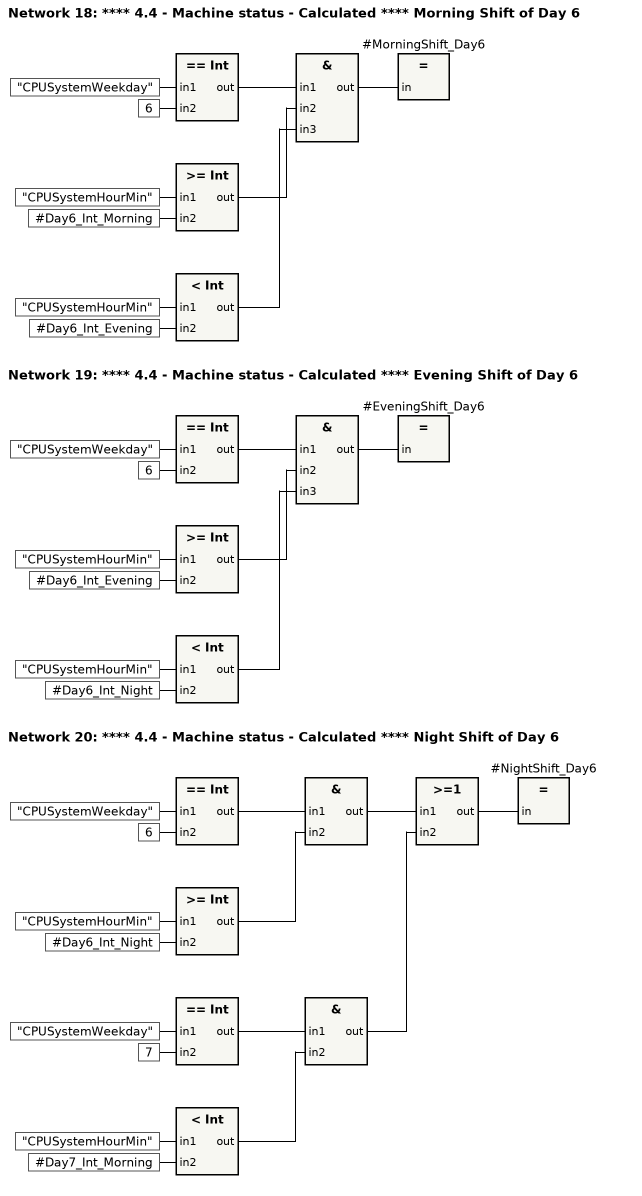
   #MorningShift_Day6 := ("CPUSystemWeekday" = 6) AND ("CPUSystemHourMin" >= #Day6_Int_Morning) AND ("CPUSystemHourMin" < #Day6_Int_Evening);
END_REGION

REGION Network 19: **** 4.4 - Machine status - Calculated **** Evening Shift of Day 6
   // Evening Shift of Day 6
   #EveningShift_Day6 := ("CPUSystemWeekday" = 6) AND ("CPUSystemHourMin" >= #Day6_Int_Evening) AND ("CPUSystemHourMin" < #Day6_Int_Night);
END_REGION

REGION Network 20: **** 4.4 - Machine status - Calculated **** Night Shift of Day 6
   // Night Shift of Day 6
   #NightShift_Day6 := (("CPUSystemWeekday" = 6) AND ("CPUSystemHourMin" >= #Day6_Int_Night)) OR (("CPUSystemWeekday" = 7) AND ("CPUSystemHourMin" < #Day7_Int_Morning));
END_REGION

REGION Network 21: **** 4.4 - Machine status - Calculated **** Morning Shift of Day 7
   // Morning Shift of Day 7
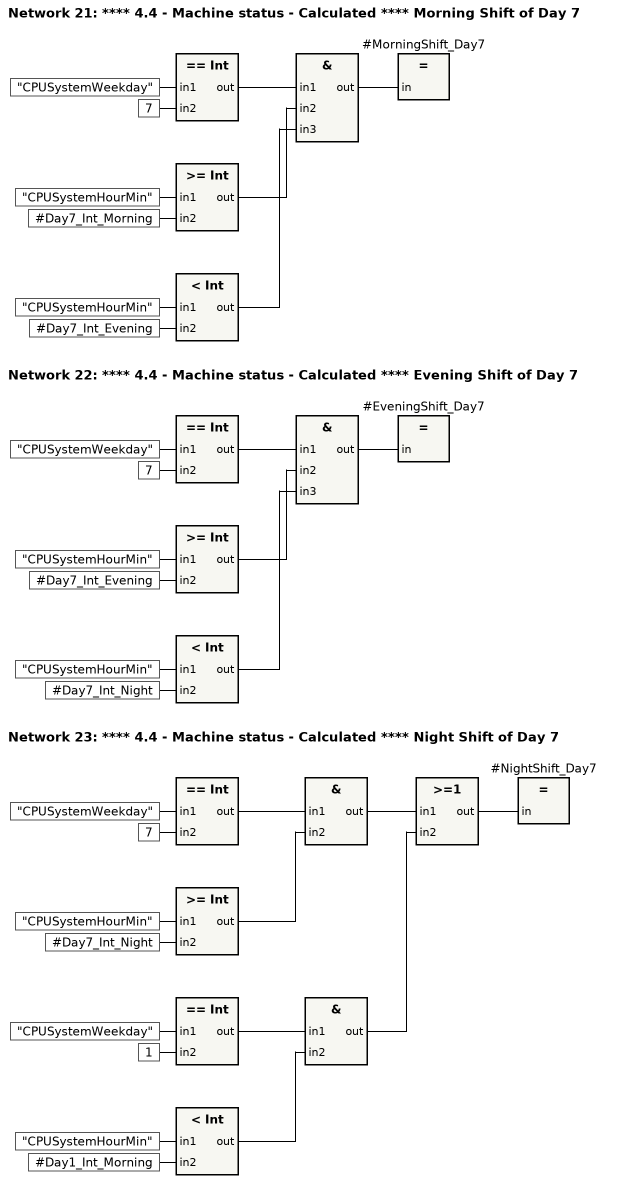
   #MorningShift_Day7 := ("CPUSystemWeekday" = 7) AND ("CPUSystemHourMin" >= #Day7_Int_Morning) AND ("CPUSystemHourMin" < #Day7_Int_Evening);
END_REGION

REGION Network 22: **** 4.4 - Machine status - Calculated **** Evening Shift of Day 7
   // Evening Shift of Day 7
   #EveningShift_Day7 := ("CPUSystemWeekday" = 7) AND ("CPUSystemHourMin" >= #Day7_Int_Evening) AND ("CPUSystemHourMin" < #Day7_Int_Night);
END_REGION

REGION Network 23: **** 4.4 - Machine status - Calculated **** Night Shift of Day 7
   // Night Shift of Day 7
   #NightShift_Day7 := (("CPUSystemWeekday" = 7) AND ("CPUSystemHourMin" >= #Day7_Int_Night)) OR (("CPUSystemWeekday" = 1) AND ("CPUSystemHourMin" < #Day1_Int_Morning));
END_REGION

REGION Network 24: **** 4.4 - Machine status - Calculated **** Morning shift
   // Morning shift
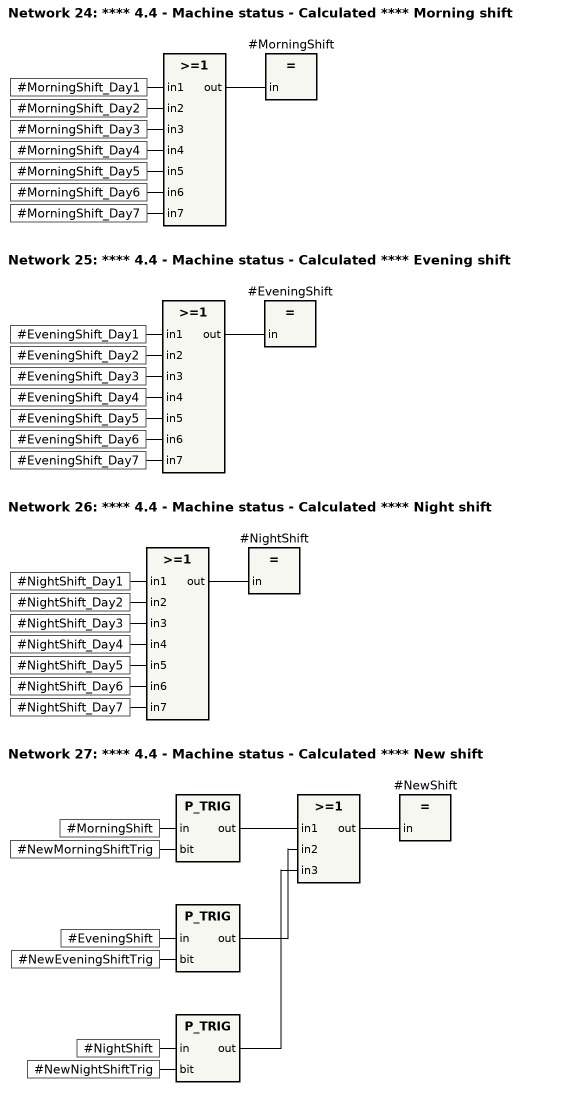
   #MorningShift := #MorningShift_Day1 OR #MorningShift_Day2 OR #MorningShift_Day3 OR #MorningShift_Day4 OR #MorningShift_Day5 OR #MorningShift_Day6 OR #MorningShift_Day7;
END_REGION

REGION Network 25: **** 4.4 - Machine status - Calculated **** Evening shift
   // Evening shift
   #EveningShift := #EveningShift_Day1 OR #EveningShift_Day2 OR #EveningShift_Day3 OR #EveningShift_Day4 OR #EveningShift_Day5 OR #EveningShift_Day6 OR #EveningShift_Day7;
END_REGION

REGION Network 26: **** 4.4 - Machine status - Calculated **** Night shift
   // Night shift
   #NightShift := #NightShift_Day1 OR #NightShift_Day2 OR #NightShift_Day3 OR #NightShift_Day4 OR #NightShift_Day5 OR #NightShift_Day6 OR #NightShift_Day7;
END_REGION

REGION Network 27: **** 4.4 - Machine status - Calculated **** New shift
   #_w1 := #MorningShift AND NOT #NewMorningShiftTrig;   // rising edge
   #NewMorningShiftTrig := #MorningShift;
   #_w2 := #EveningShift AND NOT #NewEveningShiftTrig;   // rising edge
   #NewEveningShiftTrig := #EveningShift;
   #_w3 := #NightShift AND NOT #NewNightShiftTrig;   // rising edge
   #NewNightShiftTrig := #NightShift;
   #NewShift := #_w1 OR #_w2 OR #_w3;
END_REGION

NETWORK
TITLE = **** 4.4 - Machine status - Calculated **** Days of the week
// Days of the week

//Day1
      L     "CPUSystemWeekday";
      L     1;
      ==I;
      =     #Day1;

//Day2
      L     "CPUSystemWeekday";
      L     2;
      ==I;
      =     #Day2;

//Day3
      L     "CPUSystemWeekday";
      L     3;
      ==I;
      =     #Day3;

//Day4
      L     "CPUSystemWeekday";
      L     4;
      ==I;
      =     #Day4;

//Day5
      L     "CPUSystemWeekday";
      L     5;
      ==I;
      =     #Day5;

//Day6
      L     "CPUSystemWeekday";
      L     6;
      ==I;
      =     #Day6;

//Day7
      L     "CPUSystemWeekday";
      L     7;
      ==I;
      =     #Day7;


REGION Network 29: **** 4.6 - Machine status - Indications **** Icon Animation
   // Icon Animation for HMI
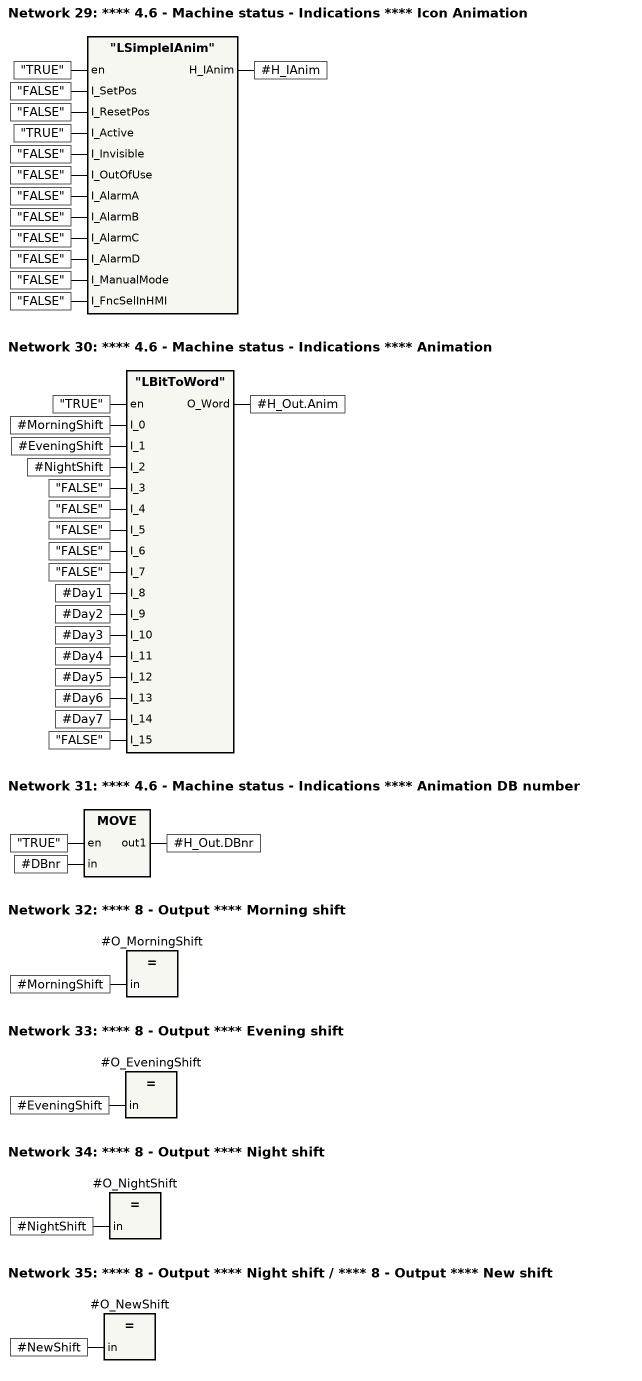
   IF "TRUE" THEN
       "LSimpleIAnim"(I_SetPos := "FALSE",
                      I_ResetPos := "FALSE",
                      I_Active := "TRUE",
                      I_Invisible := "FALSE",
                      I_OutOfUse := "FALSE",
                      I_AlarmA := "FALSE",
                      I_AlarmB := "FALSE",
                      I_AlarmC := "FALSE",
                      I_AlarmD := "FALSE",
                      I_ManualMode := "FALSE",
                      I_FncSelInHMI := "FALSE",
                      H_IAnim => #H_IAnim);
   END_IF;
END_REGION

REGION Network 30: **** 4.6 - Machine status - Indications **** Animation
   // Animation for HMI
   IF "TRUE" THEN
       "LBitToWord"(I_0 := #MorningShift,
                    I_1 := #EveningShift,
                    I_2 := #NightShift,
                    I_3 := "FALSE",
                    I_4 := "FALSE",
                    I_5 := "FALSE",
                    I_6 := "FALSE",
                    I_7 := "FALSE",
                    I_8 := #Day1,
                    I_9 := #Day2,
                    I_10 := #Day3,
                    I_11 := #Day4,
                    I_12 := #Day5,
                    I_13 := #Day6,
                    I_14 := #Day7,
                    I_15 := "FALSE",
                    O_Word => #H_Out.Anim);
   END_IF;
END_REGION

REGION Network 31: **** 4.6 - Machine status - Indications **** Animation DB number
   // Animation DB number
   IF "TRUE" THEN #H_Out.DBnr := #DBnr; END_IF;
END_REGION

REGION Network 32: **** 8 - Output **** Morning shift
   // Morning shift
   #O_MorningShift := #MorningShift;
END_REGION

REGION Network 33: **** 8 - Output **** Evening shift
   // Evening shift
   #O_EveningShift := #EveningShift;
END_REGION

REGION Network 34: **** 8 - Output **** Night shift
   // Night shift
   #O_NightShift := #NightShift;
END_REGION

REGION Network 35: **** 8 - Output **** Night shift / **** 8 - Output **** New shift
   // Night shift
   #O_NewShift := #NewShift;
END_REGION

REGION Network 36: **** 8 - Output **** Active Shift
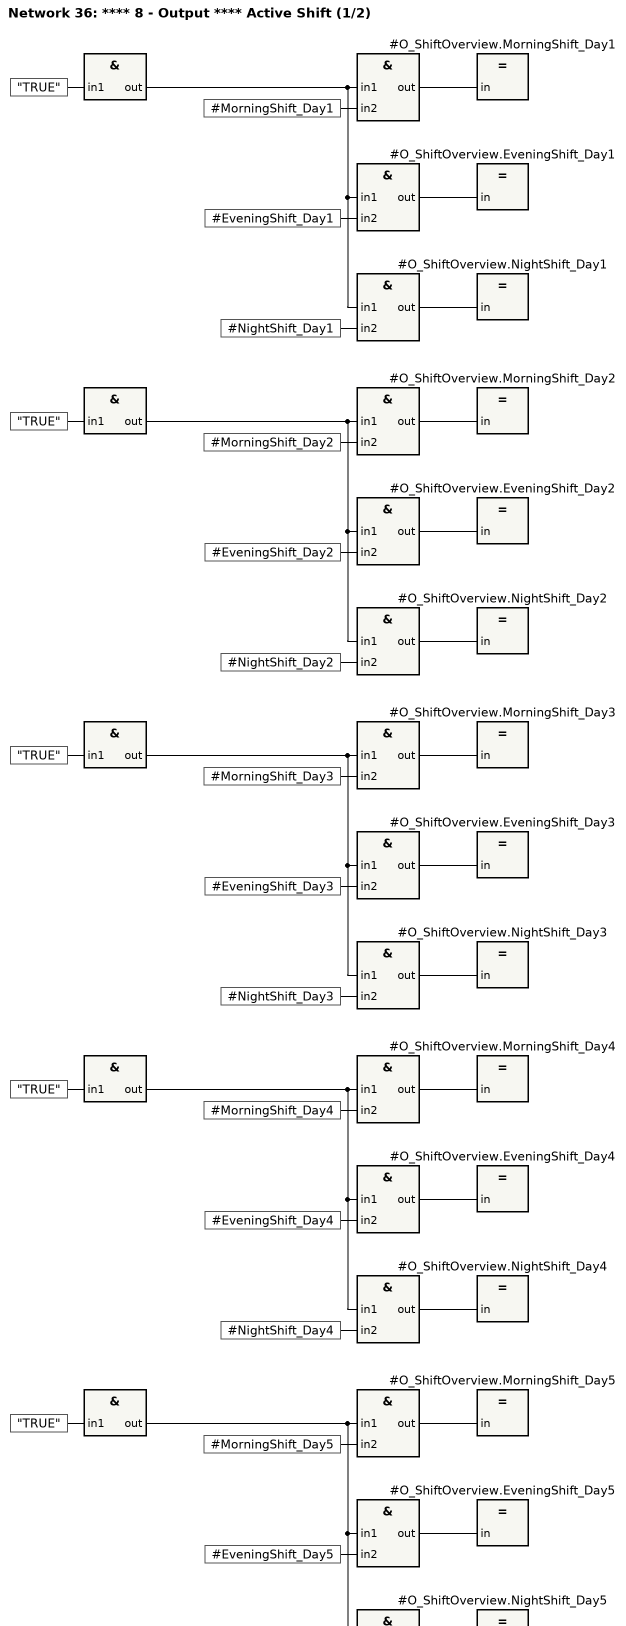
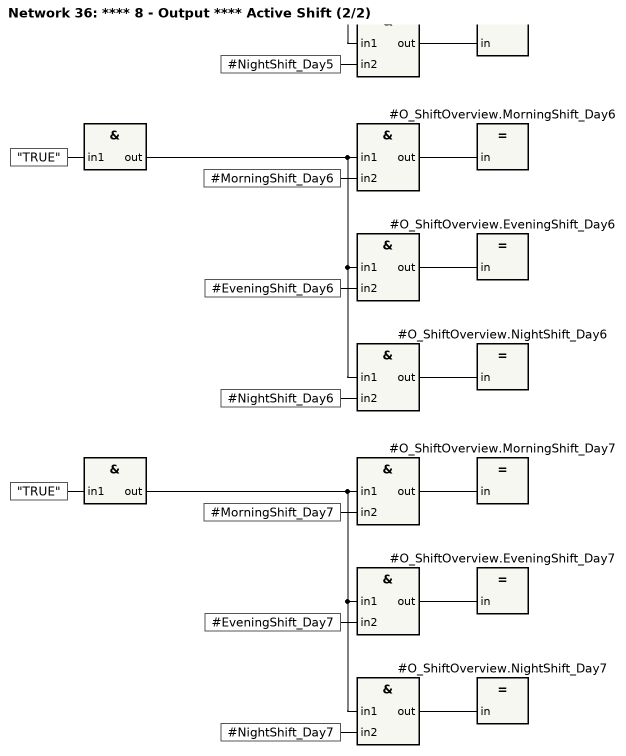
   #O_ShiftOverview.MorningShift_Day1 := "TRUE" AND #MorningShift_Day1;
   #O_ShiftOverview.EveningShift_Day1 := "TRUE" AND #EveningShift_Day1;
   #O_ShiftOverview.NightShift_Day1 := "TRUE" AND #NightShift_Day1;
   #O_ShiftOverview.MorningShift_Day2 := "TRUE" AND #MorningShift_Day2;
   #O_ShiftOverview.EveningShift_Day2 := "TRUE" AND #EveningShift_Day2;
   #O_ShiftOverview.NightShift_Day2 := "TRUE" AND #NightShift_Day2;
   #O_ShiftOverview.MorningShift_Day3 := "TRUE" AND #MorningShift_Day3;
   #O_ShiftOverview.EveningShift_Day3 := "TRUE" AND #EveningShift_Day3;
   #O_ShiftOverview.NightShift_Day3 := "TRUE" AND #NightShift_Day3;
   #O_ShiftOverview.MorningShift_Day4 := "TRUE" AND #MorningShift_Day4;
   #O_ShiftOverview.EveningShift_Day4 := "TRUE" AND #EveningShift_Day4;
   #O_ShiftOverview.NightShift_Day4 := "TRUE" AND #NightShift_Day4;
   #O_ShiftOverview.MorningShift_Day5 := "TRUE" AND #MorningShift_Day5;
   #O_ShiftOverview.EveningShift_Day5 := "TRUE" AND #EveningShift_Day5;
   #O_ShiftOverview.NightShift_Day5 := "TRUE" AND #NightShift_Day5;
   #O_ShiftOverview.MorningShift_Day6 := "TRUE" AND #MorningShift_Day6;
   #O_ShiftOverview.EveningShift_Day6 := "TRUE" AND #EveningShift_Day6;
   #O_ShiftOverview.NightShift_Day6 := "TRUE" AND #NightShift_Day6;
   #O_ShiftOverview.MorningShift_Day7 := "TRUE" AND #MorningShift_Day7;
   #O_ShiftOverview.EveningShift_Day7 := "TRUE" AND #EveningShift_Day7;
   #O_ShiftOverview.NightShift_Day7 := "TRUE" AND #NightShift_Day7;
END_REGION
END_FUNCTION_BLOCK

FUNCTION_BLOCK "LProcProdMode"   // FB1716, FBD
TITLE = LProcProductionMode
{ S7_Optimized_Access := 'FALSE' }
AUTHOR : VCC
FAMILY : Control
NAME : PrProdMo
VERSION : 1.0
// ================================================================================
// This module handles all production modes for a process modezone. The production 
// modes are Weekend, Maintenance and Production Stop.
// ================================================================================
// stored: AutoNumber false, IsIECCheckEnabled false, SetENOAutomatically False, UDAEnableTagReadback false
   VAR_INPUT
      I_ExtWeekendReq { ExternalAccessible := 'False'; ExternalVisible := 'False'; ExternalWritable := 'False'} : Bool;   // External bypass request
      I_WeekendReached { ExternalAccessible := 'False'; ExternalVisible := 'False'; ExternalWritable := 'False'} : Bool;   // Weekend reached
      I_ExtMaintReq { ExternalAccessible := 'False'; ExternalVisible := 'False'; ExternalWritable := 'False'} : Bool;   // External Maintenance request
      I_MaintReached { ExternalAccessible := 'False'; ExternalVisible := 'False'; ExternalWritable := 'False'} : Bool;   // Maintenance reached
      I_ExtProdStpReq { ExternalAccessible := 'False'; ExternalVisible := 'False'; ExternalWritable := 'False'} : Bool;   // External production stop request
      I_ProdStpReached { ExternalAccessible := 'False'; ExternalVisible := 'False'; ExternalWritable := 'False'} : Bool;   // Production mode reached
   END_VAR
   VAR_OUTPUT
      O_ProcProdMode { ExternalAccessible := 'False'; ExternalVisible := 'False'; ExternalWritable := 'False'} : Word;   // Prodution Modes
      O_WeekendModeSel { ExternalAccessible := 'False'; ExternalVisible := 'False'; ExternalWritable := 'False'} : Bool;   // Weekend mode selected
      O_WeekendMode { ExternalAccessible := 'False'; ExternalVisible := 'False'; ExternalWritable := 'False'} : Bool;   // Weekend mode active
      O_MaintModeSel { ExternalAccessible := 'False'; ExternalVisible := 'False'; ExternalWritable := 'False'} : Bool;   // Maintenance mode selected
      O_MaintMode { ExternalAccessible := 'False'; ExternalVisible := 'False'; ExternalWritable := 'False'} : Bool;   // Maintenance mode active
      O_ProdStpModeSel { ExternalAccessible := 'False'; ExternalVisible := 'False'; ExternalWritable := 'False'} : Bool;   // Production mode selected
      O_ProdStpMode { ExternalAccessible := 'False'; ExternalVisible := 'False'; ExternalWritable := 'False'} : Bool;   // Production mode active
      O_AnyProdModeSel { ExternalAccessible := 'False'; ExternalVisible := 'False'; ExternalWritable := 'False'} : Bool;   // Any production mode selected
      O_AnyProdModeActive { ExternalAccessible := 'False'; ExternalVisible := 'False'; ExternalWritable := 'False'} : Bool;   // Any production mode active
      O_AlarmABCondition { ExternalAccessible := 'False'; ExternalVisible := 'False'; ExternalWritable := 'False'} : Bool;   // Alarm AB condition
      O_AlarmA { ExternalAccessible := 'False'; ExternalVisible := 'False'; ExternalWritable := 'False'} : Bool;   // Alarms A
      O_AlarmB { ExternalAccessible := 'False'; ExternalVisible := 'False'; ExternalWritable := 'False'} : Bool;   // Alarms B
      O_AlarmC { ExternalAccessible := 'False'; ExternalVisible := 'False'; ExternalWritable := 'False'} : Bool;   // Alarms C
      O_AlarmD { ExternalAccessible := 'False'; ExternalVisible := 'False'; ExternalWritable := 'False'} : Bool;   // Alarms D
      H_AlarmWord { ExternalAccessible := 'False'; ExternalVisible := 'False'; ExternalWritable := 'False'} : DWord;   // Alarm Word
   END_VAR
   VAR DB_SPECIFIC
      AD_WESelected { ExternalAccessible := 'False'; ExternalVisible := 'False'; ExternalWritable := 'False'} : Bool;   // Week-end mode selected
      AD_MaintSelected { ExternalAccessible := 'False'; ExternalVisible := 'False'; ExternalWritable := 'False'} : Bool;   // Maintenance mode selected
      AD_ProdStopSelected { ExternalAccessible := 'False'; ExternalVisible := 'False'; ExternalWritable := 'False'} : Bool;   // Production mode selected
      H_HMIProcModeCmd : Word;   // Production mode commands from HMI
      H_Anim : Word;   // Animation
      HMIWeekendReq { ExternalAccessible := 'False'; ExternalVisible := 'False'; ExternalWritable := 'False'} : Bool;   // Bypass selected on HMI
      HMIMaintReq { ExternalAccessible := 'False'; ExternalVisible := 'False'; ExternalWritable := 'False'} : Bool;   // Maintenance selected on HMI
      HMIProdStpReq { ExternalAccessible := 'False'; ExternalVisible := 'False'; ExternalWritable := 'False'} : Bool;   // Production mode selected on HMI
      WeekendSelected { ExternalAccessible := 'False'; ExternalVisible := 'False'; ExternalWritable := 'False'} : Bool;   // Weekend is selected
      MaintSelected { ExternalAccessible := 'False'; ExternalVisible := 'False'; ExternalWritable := 'False'} : Bool;   // Maintenance is selected
      ProdStpSelected { ExternalAccessible := 'False'; ExternalVisible := 'False'; ExternalWritable := 'False'} : Bool;   // Production stop is selected
      WeekendActive { ExternalAccessible := 'False'; ExternalVisible := 'False'; ExternalWritable := 'False'} : Bool;   // Weekend is active
      MaintActive { ExternalAccessible := 'False'; ExternalVisible := 'False'; ExternalWritable := 'False'} : Bool;   // Maintenance is active
      ProdStpActive { ExternalAccessible := 'False'; ExternalVisible := 'False'; ExternalWritable := 'False'} : Bool;   // Production stop is active
      TmpMaintReqOff { ExternalAccessible := 'False'; ExternalVisible := 'False'; ExternalWritable := 'False'} : Bool;   // Temporary request off
      TmpMaintReqOn { ExternalAccessible := 'False'; ExternalVisible := 'False'; ExternalWritable := 'False'} : Bool;   // Temporary request on
      PulseMaintReqOn { ExternalAccessible := 'False'; ExternalVisible := 'False'; ExternalWritable := 'False'} : Bool;   // Pulse request on
      PulseMaintReqOff { ExternalAccessible := 'False'; ExternalVisible := 'False'; ExternalWritable := 'False'} : Bool;   // Pulse request off
      TmpWeekendReqOff { ExternalAccessible := 'False'; ExternalVisible := 'False'; ExternalWritable := 'False'} : Bool;   // Temporary request off
      TmpWeekendReqOn { ExternalAccessible := 'False'; ExternalVisible := 'False'; ExternalWritable := 'False'} : Bool;   // Temporary request on
      PulseWeekendReqOn { ExternalAccessible := 'False'; ExternalVisible := 'False'; ExternalWritable := 'False'} : Bool;   // Pulse request on
      PulseWeekendReqOff { ExternalAccessible := 'False'; ExternalVisible := 'False'; ExternalWritable := 'False'} : Bool;   // Pulse request off
      TmpProdStpReqOff { ExternalAccessible := 'False'; ExternalVisible := 'False'; ExternalWritable := 'False'} : Bool;   // Temporary request off
      TmpProdStpReqOn { ExternalAccessible := 'False'; ExternalVisible := 'False'; ExternalWritable := 'False'} : Bool;   // Temporary request on
      PulseProdStpReqOn { ExternalAccessible := 'False'; ExternalVisible := 'False'; ExternalWritable := 'False'} : Bool;   // Pulse request on
      PulseProdStpReqOff { ExternalAccessible := 'False'; ExternalVisible := 'False'; ExternalWritable := 'False'} : Bool;   // Pulse request off
      AlarmA { ExternalAccessible := 'False'; ExternalVisible := 'False'; ExternalWritable := 'False'} : Bool;   // Alarm A active in the FB
      AlarmB { ExternalAccessible := 'False'; ExternalVisible := 'False'; ExternalWritable := 'False'} : Bool;   // Alarm B active in the FB
      AlarmC { ExternalAccessible := 'False'; ExternalVisible := 'False'; ExternalWritable := 'False'} : Bool;   // Alarm C active in the FB
      AlarmD { ExternalAccessible := 'False'; ExternalVisible := 'False'; ExternalWritable := 'False'} : Bool;   // Alarm D active in the FB
   END_VAR
   VAR_TEMP   // added for the SCL form of the ladder/FBD networks
      _w1 : Bool;
      _w2 : Bool;
   END_VAR
BEGIN

REGION Network 1: **** 1 - Inputs **** Extract the production modes from HMI
   // Extract the production modes from HMI
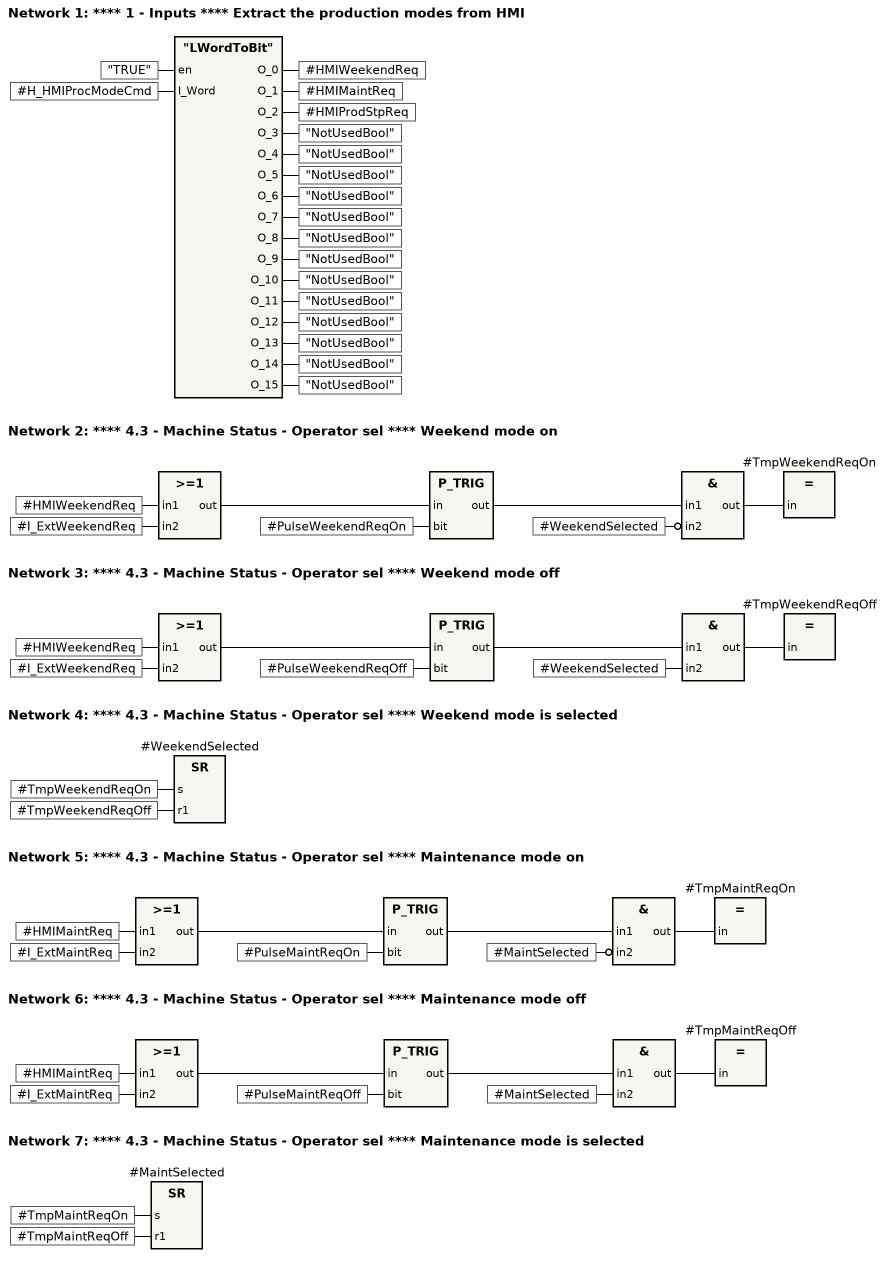
   IF "TRUE" THEN
       "LWordToBit"(I_Word := #H_HMIProcModeCmd,
                    O_0 => #HMIWeekendReq,
                    O_1 => #HMIMaintReq,
                    O_2 => #HMIProdStpReq,
                    O_3 => "NotUsedBool",
                    O_4 => "NotUsedBool",
                    O_5 => "NotUsedBool",
                    O_6 => "NotUsedBool",
                    O_7 => "NotUsedBool",
                    O_8 => "NotUsedBool",
                    O_9 => "NotUsedBool",
                    O_10 => "NotUsedBool",
                    O_11 => "NotUsedBool",
                    O_12 => "NotUsedBool",
                    O_13 => "NotUsedBool",
                    O_14 => "NotUsedBool",
                    O_15 => "NotUsedBool");
   END_IF;
END_REGION

REGION Network 2: **** 4.3 - Machine Status - Operator sel **** Weekend mode on
   // Weekend mode on
   #_w1 := #HMIWeekendReq OR #I_ExtWeekendReq;
   #_w2 := #_w1 AND NOT #PulseWeekendReqOn;   // rising edge
   #PulseWeekendReqOn := #_w1;
   #TmpWeekendReqOn := #_w2 AND NOT #WeekendSelected;
END_REGION

REGION Network 3: **** 4.3 - Machine Status - Operator sel **** Weekend mode off
   // Weekend mode off
   #_w1 := #HMIWeekendReq OR #I_ExtWeekendReq;
   #_w2 := #_w1 AND NOT #PulseWeekendReqOff;   // rising edge
   #PulseWeekendReqOff := #_w1;
   #TmpWeekendReqOff := #_w2 AND #WeekendSelected;
END_REGION

REGION Network 4: **** 4.3 - Machine Status - Operator sel **** Weekend mode is selected
   // Weekend mode is selected
   IF #TmpWeekendReqOn THEN
       #WeekendSelected := TRUE;   // SR flip-flop
   END_IF;
   IF #TmpWeekendReqOff THEN #WeekendSelected := FALSE; END_IF;
END_REGION

REGION Network 5: **** 4.3 - Machine Status - Operator sel **** Maintenance mode on
   // Maintenance mode on
   #_w1 := #HMIMaintReq OR #I_ExtMaintReq;
   #_w2 := #_w1 AND NOT #PulseMaintReqOn;   // rising edge
   #PulseMaintReqOn := #_w1;
   #TmpMaintReqOn := #_w2 AND NOT #MaintSelected;
END_REGION

REGION Network 6: **** 4.3 - Machine Status - Operator sel **** Maintenance mode off
   // Maintenance mode off
   #_w1 := #HMIMaintReq OR #I_ExtMaintReq;
   #_w2 := #_w1 AND NOT #PulseMaintReqOff;   // rising edge
   #PulseMaintReqOff := #_w1;
   #TmpMaintReqOff := #_w2 AND #MaintSelected;
END_REGION

REGION Network 7: **** 4.3 - Machine Status - Operator sel **** Maintenance mode is selected
   // Maintenance mode is selected
   IF #TmpMaintReqOn THEN
       #MaintSelected := TRUE;   // SR flip-flop
   END_IF;
   IF #TmpMaintReqOff THEN #MaintSelected := FALSE; END_IF;
END_REGION

REGION Network 8: **** 4.3 - Machine Status - Operator sel **** Production stop mode on
   // Production stop mode on
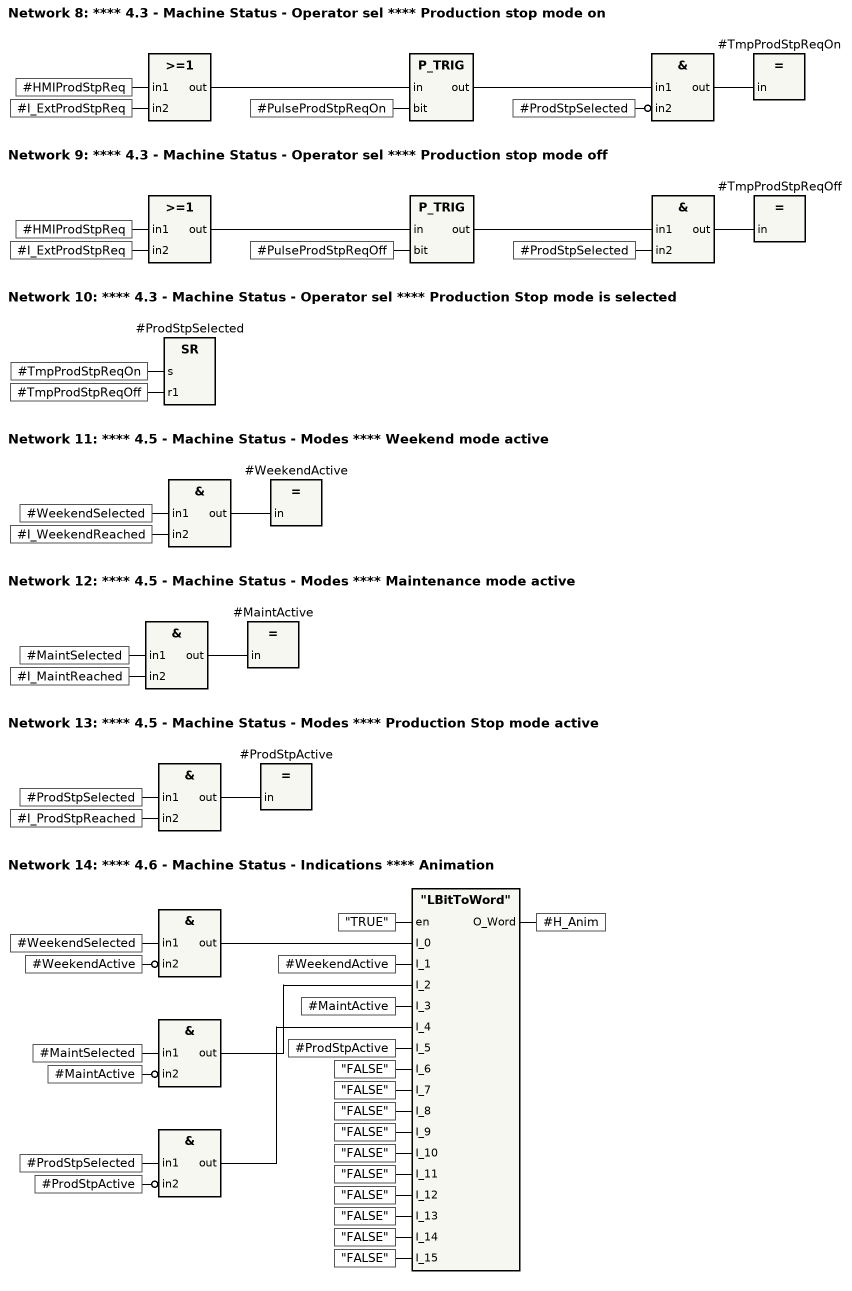
   #_w1 := #HMIProdStpReq OR #I_ExtProdStpReq;
   #_w2 := #_w1 AND NOT #PulseProdStpReqOn;   // rising edge
   #PulseProdStpReqOn := #_w1;
   #TmpProdStpReqOn := #_w2 AND NOT #ProdStpSelected;
END_REGION

REGION Network 9: **** 4.3 - Machine Status - Operator sel **** Production stop mode off
   // Production stop mode off
   #_w1 := #HMIProdStpReq OR #I_ExtProdStpReq;
   #_w2 := #_w1 AND NOT #PulseProdStpReqOff;   // rising edge
   #PulseProdStpReqOff := #_w1;
   #TmpProdStpReqOff := #_w2 AND #ProdStpSelected;
END_REGION

REGION Network 10: **** 4.3 - Machine Status - Operator sel **** Production Stop mode is selected
   // Production Stop mode is selected
   IF #TmpProdStpReqOn THEN
       #ProdStpSelected := TRUE;   // SR flip-flop
   END_IF;
   IF #TmpProdStpReqOff THEN #ProdStpSelected := FALSE; END_IF;
END_REGION

REGION Network 11: **** 4.5 - Machine Status - Modes **** Weekend mode active
   // Weekend mode active
   #WeekendActive := #WeekendSelected AND #I_WeekendReached;
END_REGION

REGION Network 12: **** 4.5 - Machine Status - Modes **** Maintenance mode active
   // Maintenance mode active
   #MaintActive := #MaintSelected AND #I_MaintReached;
END_REGION

REGION Network 13: **** 4.5 - Machine Status - Modes **** Production Stop mode active
   // Production Stop mode active
   #ProdStpActive := #ProdStpSelected AND #I_ProdStpReached;
END_REGION

REGION Network 14: **** 4.6 - Machine Status - Indications **** Animation
   // Animation
   IF "TRUE" THEN
       "LBitToWord"(I_0 := #WeekendSelected AND NOT #WeekendActive,
                    I_1 := #WeekendActive,
                    I_2 := #MaintSelected AND NOT #MaintActive,
                    I_3 := #MaintActive,
                    I_4 := #ProdStpSelected AND NOT #ProdStpActive,
                    I_5 := #ProdStpActive,
                    I_6 := "FALSE",
                    I_7 := "FALSE",
                    I_8 := "FALSE",
                    I_9 := "FALSE",
                    I_10 := "FALSE",
                    I_11 := "FALSE",
                    I_12 := "FALSE",
                    I_13 := "FALSE",
                    I_14 := "FALSE",
                    I_15 := "FALSE",
                    O_Word => #H_Anim);
   END_IF;
END_REGION

REGION Network 15: **** 8 - Outputs **** Set the different bits in the Production Mode register
   // Set the different bits in the Production Mode register
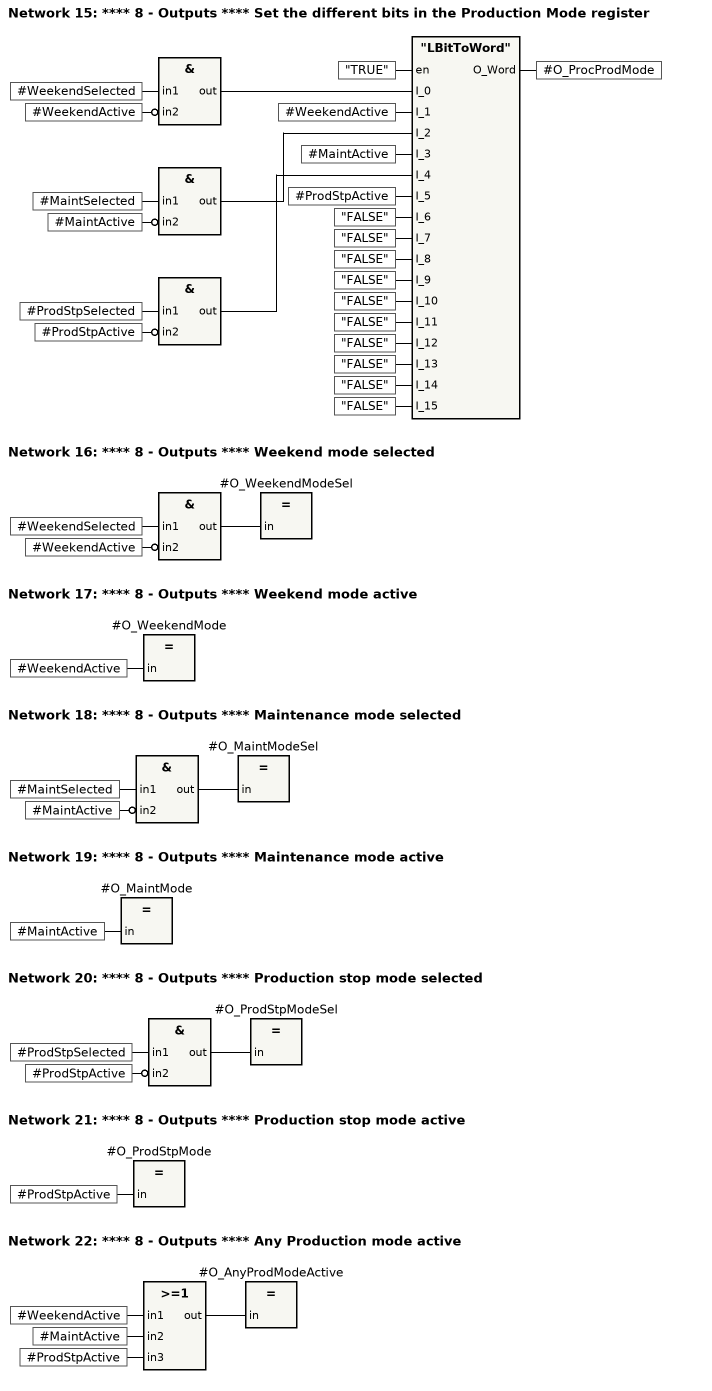
   IF "TRUE" THEN
       "LBitToWord"(I_0 := #WeekendSelected AND NOT #WeekendActive,
                    I_1 := #WeekendActive,
                    I_2 := #MaintSelected AND NOT #MaintActive,
                    I_3 := #MaintActive,
                    I_4 := #ProdStpSelected AND NOT #ProdStpActive,
                    I_5 := #ProdStpActive,
                    I_6 := "FALSE",
                    I_7 := "FALSE",
                    I_8 := "FALSE",
                    I_9 := "FALSE",
                    I_10 := "FALSE",
                    I_11 := "FALSE",
                    I_12 := "FALSE",
                    I_13 := "FALSE",
                    I_14 := "FALSE",
                    I_15 := "FALSE",
                    O_Word => #O_ProcProdMode);
   END_IF;
END_REGION

REGION Network 16: **** 8 - Outputs **** Weekend mode selected
   // Weekend mode selected
   #O_WeekendModeSel := #WeekendSelected AND NOT #WeekendActive;
END_REGION

REGION Network 17: **** 8 - Outputs **** Weekend mode active
   // Weekend mode active
   #O_WeekendMode := #WeekendActive;
END_REGION

REGION Network 18: **** 8 - Outputs **** Maintenance mode selected
   // Maintenance mode selected
   #O_MaintModeSel := #MaintSelected AND NOT #MaintActive;
END_REGION

REGION Network 19: **** 8 - Outputs **** Maintenance mode active
   // Maintenance mode active
   #O_MaintMode := #MaintActive;
END_REGION

REGION Network 20: **** 8 - Outputs **** Production stop mode selected
   // Production stop mode selected
   #O_ProdStpModeSel := #ProdStpSelected AND NOT #ProdStpActive;
END_REGION

REGION Network 21: **** 8 - Outputs **** Production stop mode active
   // Production stop mode active
   #O_ProdStpMode := #ProdStpActive;
END_REGION

REGION Network 22: **** 8 - Outputs **** Any Production mode active
   // Any Production mode active
   #O_AnyProdModeActive := #WeekendActive OR #MaintActive OR #ProdStpActive;
END_REGION

REGION Network 23: **** 8 - Outputs **** Any Production mode active
   // Any Production mode active
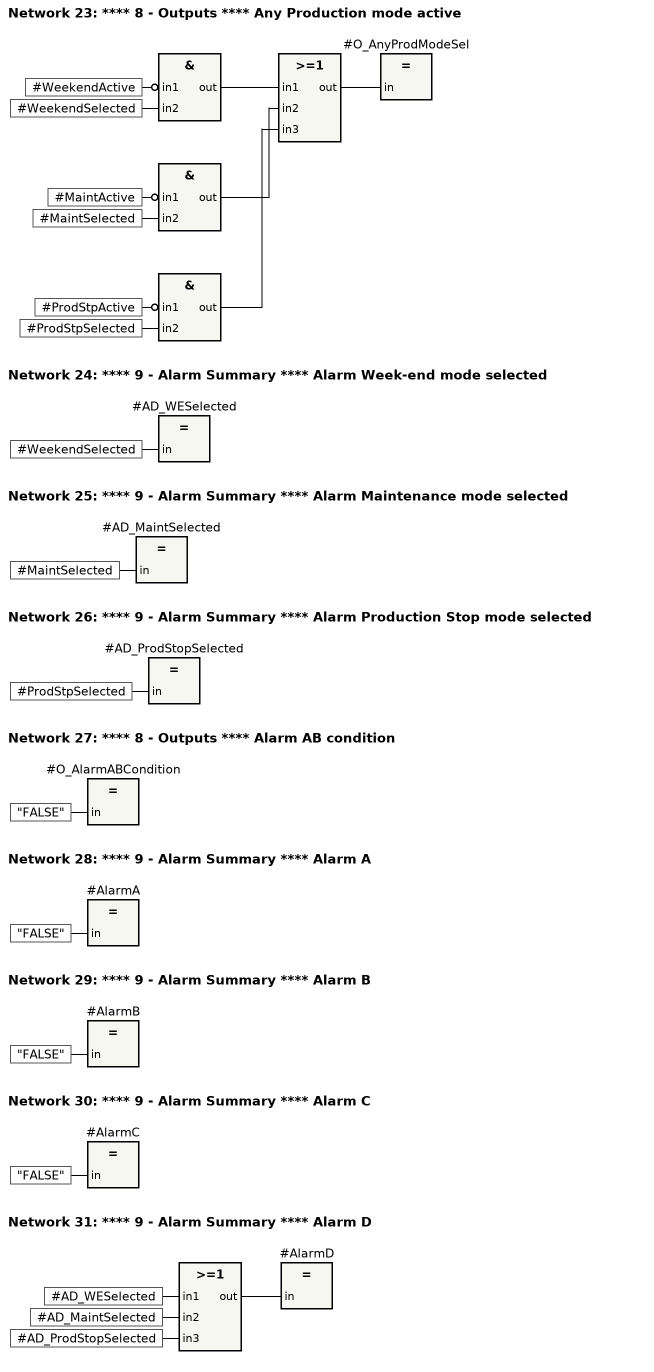
   #O_AnyProdModeSel := (NOT #WeekendActive AND #WeekendSelected) OR (NOT #MaintActive AND #MaintSelected) OR (NOT #ProdStpActive AND #ProdStpSelected);
END_REGION

REGION Network 24: **** 9 - Alarm Summary **** Alarm Week-end mode selected
   // Alarm Week-end mode selected
   #AD_WESelected := #WeekendSelected;
END_REGION

REGION Network 25: **** 9 - Alarm Summary **** Alarm Maintenance mode selected
   // Alarm Maintenance mode selected
   #AD_MaintSelected := #MaintSelected;
END_REGION

REGION Network 26: **** 9 - Alarm Summary **** Alarm Production Stop mode selected
   // Alarm Production Stop mode selected
   #AD_ProdStopSelected := #ProdStpSelected;
END_REGION

REGION Network 27: **** 8 - Outputs **** Alarm AB condition
   // Alarm AB condition
   #O_AlarmABCondition := "FALSE";
END_REGION

REGION Network 28: **** 9 - Alarm Summary **** Alarm A
   // Summary of alarms A
   #AlarmA := "FALSE";
END_REGION

REGION Network 29: **** 9 - Alarm Summary **** Alarm B
   // Summary of alarms B
   #AlarmB := "FALSE";
END_REGION

REGION Network 30: **** 9 - Alarm Summary **** Alarm C
   // Summary of alarms C
   #AlarmC := "FALSE";
END_REGION

REGION Network 31: **** 9 - Alarm Summary **** Alarm D
   // Summary of alarms D
   #AlarmD := #AD_WESelected OR #AD_MaintSelected OR #AD_ProdStopSelected;
END_REGION

REGION Network 32: **** 9.1 - Alarm Output **** Alarm A
   // Summary of alarms A
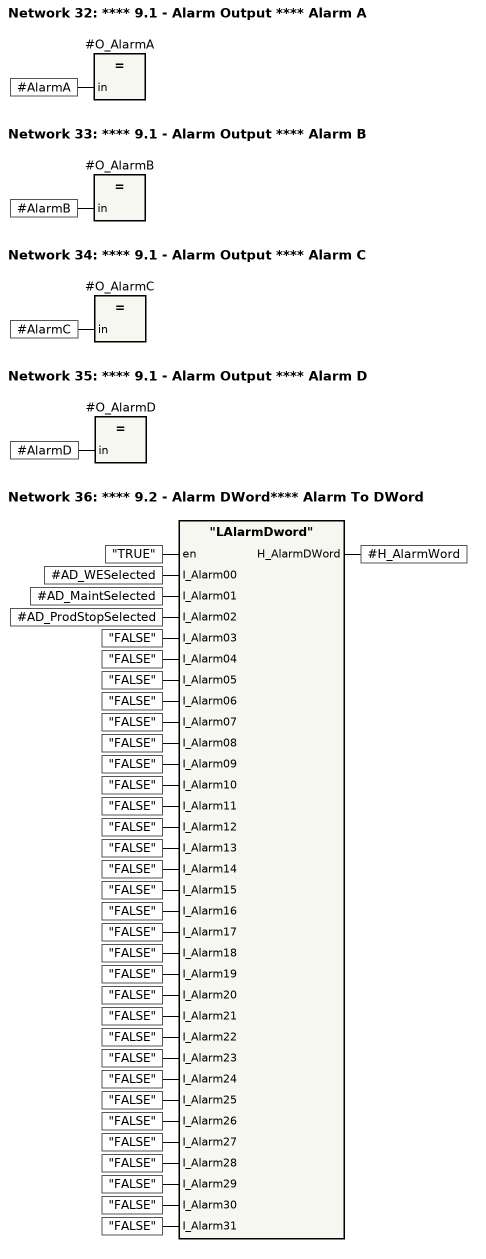
   #O_AlarmA := #AlarmA;
END_REGION

REGION Network 33: **** 9.1 - Alarm Output **** Alarm B
   // Summary of alarms B
   #O_AlarmB := #AlarmB;
END_REGION

REGION Network 34: **** 9.1 - Alarm Output **** Alarm C
   // Summary of alarms C
   #O_AlarmC := #AlarmC;
END_REGION

REGION Network 35: **** 9.1 - Alarm Output **** Alarm D
   // Summary of alarms D
   #O_AlarmD := #AlarmD;
END_REGION

REGION Network 36: **** 9.2 - Alarm DWord**** Alarm To DWord
   // Alarm Word
   IF "TRUE" THEN
       "LAlarmDword"(I_Alarm00 := #AD_WESelected,
                     I_Alarm01 := #AD_MaintSelected,
                     I_Alarm02 := #AD_ProdStopSelected,
                     I_Alarm03 := "FALSE",
                     I_Alarm04 := "FALSE",
                     I_Alarm05 := "FALSE",
                     I_Alarm06 := "FALSE",
                     I_Alarm07 := "FALSE",
                     I_Alarm08 := "FALSE",
                     I_Alarm09 := "FALSE",
                     I_Alarm10 := "FALSE",
                     I_Alarm11 := "FALSE",
                     I_Alarm12 := "FALSE",
                     I_Alarm13 := "FALSE",
                     I_Alarm14 := "FALSE",
                     I_Alarm15 := "FALSE",
                     I_Alarm16 := "FALSE",
                     I_Alarm17 := "FALSE",
                     I_Alarm18 := "FALSE",
                     I_Alarm19 := "FALSE",
                     I_Alarm20 := "FALSE",
                     I_Alarm21 := "FALSE",
                     I_Alarm22 := "FALSE",
                     I_Alarm23 := "FALSE",
                     I_Alarm24 := "FALSE",
                     I_Alarm25 := "FALSE",
                     I_Alarm26 := "FALSE",
                     I_Alarm27 := "FALSE",
                     I_Alarm28 := "FALSE",
                     I_Alarm29 := "FALSE",
                     I_Alarm30 := "FALSE",
                     I_Alarm31 := "FALSE",
                     H_AlarmDWord => #H_AlarmWord);
   END_IF;
END_REGION
END_FUNCTION_BLOCK

FUNCTION_BLOCK "LMode"   // FB1000, FBD
TITLE = LMode
{ S7_Optimized_Access := 'FALSE' }
AUTHOR : VCC
FAMILY : Control
NAME : Mode
VERSION : 1.0
// ================================================================================
// This module is used to handle all operating modes for a modezone as well as 
// resetting of alarms. It get the input from LModeSelector.
// ================================================================================
// stored: AutoNumber false, IsIECCheckEnabled false, SetENOAutomatically False, UDAEnableTagReadback false
   VAR_INPUT
      I_NormalStop { ExternalAccessible := 'False'; ExternalVisible := 'False'; ExternalWritable := 'False'} : Bool;   // Normal Stop Activated Stop Automatic
      I_EnableAlarms { ExternalAccessible := 'False'; ExternalVisible := 'False'; ExternalWritable := 'False'} : Bool;   // Filter alarms for lower levels
      I_AutoModeSel { ExternalAccessible := 'False'; ExternalVisible := 'False'; ExternalWritable := 'False'} : Bool;   // Auto selected
      I_StepModeSel { ExternalAccessible := 'False'; ExternalVisible := 'False'; ExternalWritable := 'False'} : Bool;   // Step selected
      I_HomeRunModeSel { ExternalAccessible := 'False'; ExternalVisible := 'False'; ExternalWritable := 'False'} : Bool;   // Homerun selected
      I_HomeRunPush { ExternalAccessible := 'False'; ExternalVisible := 'False'; ExternalWritable := 'False'} : Bool;   // The reset button needs to be active during the homerun
      I_ManualModeSel { ExternalAccessible := 'False'; ExternalVisible := 'False'; ExternalWritable := 'False'} : Bool;   // Manual selected
      I_ForcedManActSel { ExternalAccessible := 'False'; ExternalVisible := 'False'; ExternalWritable := 'False'} : Bool;   // Forced manual key switch
      I_HomerunCond { ExternalAccessible := 'False'; ExternalVisible := 'False'; ExternalWritable := 'False'} : Bool;   // Condition for homerun
      I_HomePos { ExternalAccessible := 'False'; ExternalVisible := 'False'; ExternalWritable := 'False'} : Bool;   // Station in homposition
      I_AfterHomerunSel { ExternalAccessible := 'False'; ExternalVisible := 'False'; ExternalWritable := 'False'} : Bool;   // Show selection after Homrun on HMI
      I_HomeRunRedoSel { ExternalAccessible := 'False'; ExternalVisible := 'False'; ExternalWritable := 'False'} : Bool;   // Redo after Homerun selected
      I_HomeRunWorkDoneSel { ExternalAccessible := 'False'; ExternalVisible := 'False'; ExternalWritable := 'False'} : Bool;   // WorkDone after Homerun selected
      I_HomeRunRedoReset { ExternalAccessible := 'False'; ExternalVisible := 'False'; ExternalWritable := 'False'} : Bool;   // Reset redo after homerun
      I_HomeRunWorkDoneReset { ExternalAccessible := 'False'; ExternalVisible := 'False'; ExternalWritable := 'False'} : Bool;   // Reset workdone after homerun
      I_HomeRunPriorityRedo { ExternalAccessible := 'False'; ExternalVisible := 'False'; ExternalWritable := 'False'} : Bool;   // Priority Redo after homerun
      I_CycleFinishedSel { ExternalAccessible := 'False'; ExternalVisible := 'False'; ExternalWritable := 'False'} : Bool;   // Cycle finished is selected
      I_StartPBSel { ExternalAccessible := 'False'; ExternalVisible := 'False'; ExternalWritable := 'False'} : Bool;   // Summary of Start buttons
      I_AlarmResetPBSel { ExternalAccessible := 'False'; ExternalVisible := 'False'; ExternalWritable := 'False'} : Bool;   // Summary of Alarm reset buttons
      I_PBSetSel { ExternalAccessible := 'False'; ExternalVisible := 'False'; ExternalWritable := 'False'} : Bool;   // Pushbutton Set
      I_PBResetSel { ExternalAccessible := 'False'; ExternalVisible := 'False'; ExternalWritable := 'False'} : Bool;   // Pushbutton Reset
      I_ResetSeqSel { ExternalAccessible := 'False'; ExternalVisible := 'False'; ExternalWritable := 'False'} : Bool;   // Reset Sequence
      I_ResetTMSel { ExternalAccessible := 'False'; ExternalVisible := 'False'; ExternalWritable := 'False'} : Bool;   // Reset Transport memory
      I_SafetyOk { ExternalAccessible := 'False'; ExternalVisible := 'False'; ExternalWritable := 'False'} : Bool;   // SafetyOk / No Haltbutton is activate
      I_NotHaltButton { ExternalAccessible := 'False'; ExternalVisible := 'False'; ExternalWritable := 'False'} : Bool;   // No Haltbutton is activate
      I_ExtAutoCond { ExternalAccessible := 'False'; ExternalVisible := 'False'; ExternalWritable := 'False'} : Bool;   // External Auto Conditions / No Haltbutton is activate
      I_AlarmABCondition { ExternalAccessible := 'False'; ExternalVisible := 'False'; ExternalWritable := 'False'} : Bool;   // Alarm AB condition in the Modezone / Alarm AB condition
      I_AlarmA { ExternalAccessible := 'False'; ExternalVisible := 'False'; ExternalWritable := 'False'} : Bool;   // Alarm A active in the Modezone / Alarm A active in the modezone
      I_AlarmB { ExternalAccessible := 'False'; ExternalVisible := 'False'; ExternalWritable := 'False'} : Bool;   // Alarm B active in the Modezone / Alarm B active in the modezone
      I_AlarmC { ExternalAccessible := 'False'; ExternalVisible := 'False'; ExternalWritable := 'False'} : Bool;   // Alarm C active in the Modezone / Alarm C active in the modezone
      I_AlarmD { ExternalAccessible := 'False'; ExternalVisible := 'False'; ExternalWritable := 'False'} : Bool;   // Alarm D active in the Modezone
      I_UpperLevelZSAlarmABCondition { ExternalAccessible := 'False'; ExternalVisible := 'False'; ExternalWritable := 'False'} : Bool;   // Alarm AB condition from the Safety Zone / Alarm AB condition
      I_UpperLevelZSAlarmA { ExternalAccessible := 'False'; ExternalVisible := 'False'; ExternalWritable := 'False'} : Bool;   // Alarm A active from the Safety Zone / Alarm A active from the top level
      I_UpperLevelZSAlarmB { ExternalAccessible := 'False'; ExternalVisible := 'False'; ExternalWritable := 'False'} : Bool;   // Alarm B active from the Safety Zone / Alarm B active from the top level
      I_UpperLevelZSAlarmC { ExternalAccessible := 'False'; ExternalVisible := 'False'; ExternalWritable := 'False'} : Bool;   // Alarm C active from the Safety Zone / Alarm C active from the top level
      I_UpperLevelZSAlarmD { ExternalAccessible := 'False'; ExternalVisible := 'False'; ExternalWritable := 'False'} : Bool;   // Alarm D active from the Safety Zone
      I_UpperLevelPLCAlarmABCondition { ExternalAccessible := 'False'; ExternalVisible := 'False'; ExternalWritable := 'False'} : Bool;   // Alarm AB condition from the PLC level / Alarm AB condition
      I_UpperLevelPLCAlarmA { ExternalAccessible := 'False'; ExternalVisible := 'False'; ExternalWritable := 'False'} : Bool;   // Alarm A active from the PLC level / Alarm A active from the top level
      I_UpperLevelPLCAlarmB { ExternalAccessible := 'False'; ExternalVisible := 'False'; ExternalWritable := 'False'} : Bool;   // Alarm B active from the PLC level / Alarm B active from the top level
      I_UpperLevelPLCAlarmC { ExternalAccessible := 'False'; ExternalVisible := 'False'; ExternalWritable := 'False'} : Bool;   // Alarm C active from the PLC level / Alarm C active from the top level
      I_UpperLevelPLCAlarmD { ExternalAccessible := 'False'; ExternalVisible := 'False'; ExternalWritable := 'False'} : Bool;   // Alarm D active from the PLC level
      I_AutoModeWarningTime { ExternalAccessible := 'False'; ExternalVisible := 'False'; ExternalWritable := 'False'} : Int;   // Auto Mode warning time / Auto mode warning time
   END_VAR
   VAR_OUTPUT
      O_AutoMode { ExternalAccessible := 'False'; ExternalVisible := 'False'; ExternalWritable := 'False'} : Bool;   // Auto Mode / Auto mode
      O_StepMode { ExternalAccessible := 'False'; ExternalVisible := 'False'; ExternalWritable := 'False'} : Bool;   // Step Mode / Step mode
      O_HomeRunMode { ExternalAccessible := 'False'; ExternalVisible := 'False'; ExternalWritable := 'False'} : Bool;   // Homrun Mode / Homrun mode
      O_ManualMode { ExternalAccessible := 'False'; ExternalVisible := 'False'; ExternalWritable := 'False'} : Bool;   // Manual Mode / Manual mode
      O_ForcedMan { ExternalAccessible := 'False'; ExternalVisible := 'False'; ExternalWritable := 'False'} : Bool;   // Forced manual
      O_AutoStepRun { ExternalAccessible := 'False'; ExternalVisible := 'False'; ExternalWritable := 'False'} : Bool;   // Auto Mode or Step Mode and StartPB is active / Auto mode or Step mode and StartPB is active
      O_AutoStepHomeRunAct { ExternalAccessible := 'False'; ExternalVisible := 'False'; ExternalWritable := 'False'} : Bool;   // Auto, Step or Homerun Mode is active / Auto, Step or Homerun mode is active
      O_StartPB { ExternalAccessible := 'False'; ExternalVisible := 'False'; ExternalWritable := 'False'} : Bool;   // Start button is activated
      O_AlarmResetPB { ExternalAccessible := 'False'; ExternalVisible := 'False'; ExternalWritable := 'False'} : Bool;   // Alarm reset button is activated
      O_SetPBMan { ExternalAccessible := 'False'; ExternalVisible := 'False'; ExternalWritable := 'False'} : Bool;   // Set pushbutton is activated in manual
      O_ResetPBMan { ExternalAccessible := 'False'; ExternalVisible := 'False'; ExternalWritable := 'False'} : Bool;   // Reset pushbutton is activated in manual
      O_ResetTM { ExternalAccessible := 'False'; ExternalVisible := 'False'; ExternalWritable := 'False'} : Bool;   // Reset transport memory
      O_ResetSeq { ExternalAccessible := 'False'; ExternalVisible := 'False'; ExternalWritable := 'False'} : Bool;   // Reset sequence
      O_CycleFinished { ExternalAccessible := 'False'; ExternalVisible := 'False'; ExternalWritable := 'False'} : Bool;   // Cycle finished
      O_AlarmABAct { ExternalAccessible := 'False'; ExternalVisible := 'False'; ExternalWritable := 'False'} : Bool;   // A or B alarm active
      O_HaltButton { ExternalAccessible := 'False'; ExternalVisible := 'False'; ExternalWritable := 'False'} : Bool;   // A Haltbutton is activated
      O_AutoModeWarning { ExternalAccessible := 'False'; ExternalVisible := 'False'; ExternalWritable := 'False'} : Bool;   // Auto Mode warning / Auto mode warning
      O_HomeRunRedo { ExternalAccessible := 'False'; ExternalVisible := 'False'; ExternalWritable := 'False'} : Bool;   // Redo work after homerun
      O_HomeRunWorkDone { ExternalAccessible := 'False'; ExternalVisible := 'False'; ExternalWritable := 'False'} : Bool;   // WorkDone after homerun
      O_HMIResetPBRedColor { ExternalAccessible := 'False'; ExternalVisible := 'False'; ExternalWritable := 'False'} : Bool;   // Red background color for the Reset button on the HMI
      O_ActiveMode : Word;   // Active Mode / Active mode
      O_SelectedMode : Word;   // Selected Mode. Only active when a Mode is selected but not started / Selected mode. Only active when a mode is selected but not started
      O_AlarmABCondition { ExternalAccessible := 'False'; ExternalVisible := 'False'; ExternalWritable := 'False'} : Bool;   // Alarm AB condition
      O_AlarmA { ExternalAccessible := 'False'; ExternalVisible := 'False'; ExternalWritable := 'False'} : Bool;   // Alarms A
      O_AlarmB { ExternalAccessible := 'False'; ExternalVisible := 'False'; ExternalWritable := 'False'} : Bool;   // Alarms B
      O_AlarmC { ExternalAccessible := 'False'; ExternalVisible := 'False'; ExternalWritable := 'False'} : Bool;   // Alarms C
      O_AlarmD { ExternalAccessible := 'False'; ExternalVisible := 'False'; ExternalWritable := 'False'} : Bool;   // Alarms D
      H_AlarmWord { ExternalAccessible := 'False'; ExternalVisible := 'False'; ExternalWritable := 'False'} : DWord;   // Alarm Word
   END_VAR
   VAR_IN_OUT
      IO_Modes : "Modes";
   END_VAR
   VAR DB_SPECIFIC
      AC_HomeRun { ExternalAccessible := 'False'; ExternalVisible := 'False'; ExternalWritable := 'False'} : Bool;   // Homerun alarm
      AC_AutoNotStarted { ExternalAccessible := 'False'; ExternalVisible := 'False'; ExternalWritable := 'False'} : Bool;   // Auto not started
      AC_StartPBSticking { ExternalAccessible := 'False'; ExternalVisible := 'False'; ExternalWritable := 'False'} : Bool;   // Start push button is ON longer then 20 sec
      AC_ResetPBSticking { ExternalAccessible := 'False'; ExternalVisible := 'False'; ExternalWritable := 'False'} : Bool;   // Reset Alarm push button is ON longer then 20 sec
      AD_ManualMode { ExternalAccessible := 'False'; ExternalVisible := 'False'; ExternalWritable := 'False'} : Bool;   // Manual Mode activated / Manual mode activated
      AD_StepModeSel { ExternalAccessible := 'False'; ExternalVisible := 'False'; ExternalWritable := 'False'} : Bool;   // Step Mode selected / Step mode selected
      AD_HomeRunMode { ExternalAccessible := 'False'; ExternalVisible := 'False'; ExternalWritable := 'False'} : Bool;   // Homerun Mode activated / Homerun mode activated
      AE_NormalStop { ExternalAccessible := 'False'; ExternalVisible := 'False'; ExternalWritable := 'False'} : Bool;   // Normal Stop Mode Activated / Normal Stop Mode activated / NormalStop Aktiverat
      AE_ResetSeq { ExternalAccessible := 'False'; ExternalVisible := 'False'; ExternalWritable := 'False'} : Bool;   // Reset sequence activated
      AE_ResetTM { ExternalAccessible := 'False'; ExternalVisible := 'False'; ExternalWritable := 'False'} : Bool;   // Reset Transport memory activated
      AE_ForcedMan { ExternalAccessible := 'False'; ExternalVisible := 'False'; ExternalWritable := 'False'} : Bool;   // Manual Forced activated
      H_Anim : Word;   // Animation
      H_Anim2 : Word;   // Animation
      H_HomeRunModeAnim : Word;   // Homerun Animation
      H_ConfigBtnResetTM : Bool;   // From the HMI - Config internal tag
      H_ConfigBtnResetSeq : Bool;   // From the HMI - Config internal tag
      H_ModeChanged : Bool;   // From the HMI - Mode changed to Auto
      H_ScreenChanged : Bool;   // From the HMI - The screen has changed
      HomeRunHold { ExternalAccessible := 'False'; ExternalVisible := 'False'; ExternalWritable := 'False'} : Bool;   // Homerun, the operator have to hold the button
      HomeRunMc { ExternalAccessible := 'False'; ExternalVisible := 'False'; ExternalWritable := 'False'} : Bool;   // Homerun without hold function
      AlarmA { ExternalAccessible := 'False'; ExternalVisible := 'False'; ExternalWritable := 'False'} : Bool;   // Alarm A active in the FB
      AlarmB { ExternalAccessible := 'False'; ExternalVisible := 'False'; ExternalWritable := 'False'} : Bool;   // Alarm B active in the FB
      AlarmC { ExternalAccessible := 'False'; ExternalVisible := 'False'; ExternalWritable := 'False'} : Bool;   // Alarm C active in the FB
      AlarmD { ExternalAccessible := 'False'; ExternalVisible := 'False'; ExternalWritable := 'False'} : Bool;   // Alarm D active in the FB
      StepPulse { ExternalAccessible := 'False'; ExternalVisible := 'False'; ExternalWritable := 'False'} : Bool;   // Step pulse
      AutoMode { ExternalAccessible := 'False'; ExternalVisible := 'False'; ExternalWritable := 'False'} : Bool;   // Auto Mode / Auto mode
      StepMode { ExternalAccessible := 'False'; ExternalVisible := 'False'; ExternalWritable := 'False'} : Bool;   // Step Mode / Step mode
      HomeRunMode { ExternalAccessible := 'False'; ExternalVisible := 'False'; ExternalWritable := 'False'} : Bool;   // Homrun Mode / Homrun mode
      ManualMode { ExternalAccessible := 'False'; ExternalVisible := 'False'; ExternalWritable := 'False'} : Bool;   // Manual Mode / Manual mode
      ForcedMan { ExternalAccessible := 'False'; ExternalVisible := 'False'; ExternalWritable := 'False'} : Bool;   // Forced manual
      AutoStepRun { ExternalAccessible := 'False'; ExternalVisible := 'False'; ExternalWritable := 'False'} : Bool;   // Auto Mode or Step Mode and StartPB is active / Auto mode or Step mode and StartPB is active
      AutoStepHomeRunAct { ExternalAccessible := 'False'; ExternalVisible := 'False'; ExternalWritable := 'False'} : Bool;   // Auto, Step or Homerun Mode is active / Auto, Step or Homerun mode is active
      SetPBMan { ExternalAccessible := 'False'; ExternalVisible := 'False'; ExternalWritable := 'False'} : Bool;   // Set pushbutton is activated in manual
      ResetPBMan { ExternalAccessible := 'False'; ExternalVisible := 'False'; ExternalWritable := 'False'} : Bool;   // Reset pushbutton is activated in manual
      ResetTM { ExternalAccessible := 'False'; ExternalVisible := 'False'; ExternalWritable := 'False'} : Bool;   // Reset transport memory
      ResetSeq { ExternalAccessible := 'False'; ExternalVisible := 'False'; ExternalWritable := 'False'} : Bool;   // Reset sequence
      HomeRunAlmCond { ExternalAccessible := 'False'; ExternalVisible := 'False'; ExternalWritable := 'False'} : Bool;   // Homerun alarm condition
      HomeRunRedo { ExternalAccessible := 'False'; ExternalVisible := 'False'; ExternalWritable := 'False'} : Bool;   // Redo work after homerun
      HomeRunWorkDone { ExternalAccessible := 'False'; ExternalVisible := 'False'; ExternalWritable := 'False'} : Bool;   // WorkDone after homerun
      HomeRunModeNegEdge1 { ExternalAccessible := 'False'; ExternalVisible := 'False'; ExternalWritable := 'False'} : Bool;   // Negative edge of homerun active
      HomeRunModeNegEdge2 { ExternalAccessible := 'False'; ExternalVisible := 'False'; ExternalWritable := 'False'} : Bool;   // Negative edge of homerun active
      HomeRunModePosEdge1 { ExternalAccessible := 'False'; ExternalVisible := 'False'; ExternalWritable := 'False'} : Bool;   // Positive edge of homerun active
      HomeRunModePosEdge2 { ExternalAccessible := 'False'; ExternalVisible := 'False'; ExternalWritable := 'False'} : Bool;   // Positive edge of homerun active
      AutoModeWarningTimer { ExternalAccessible := 'False'; ExternalVisible := 'False'; ExternalWritable := 'False'} : Bool;   // Auto Mode warning timer / Auto mode warning timer
      TimerResetSeq { ExternalAccessible := 'False'; ExternalVisible := 'False'; ExternalWritable := 'False'} : Bool;   // Timer for reset sequence
      TimerResetTM { ExternalAccessible := 'False'; ExternalVisible := 'False'; ExternalWritable := 'False'} : Bool;   // Timer for reset TM
      AutoModeWarning { ExternalAccessible := 'False'; ExternalVisible := 'False'; ExternalWritable := 'False'} : Bool;   // Auto Mode warning / Auto mode warning
      AutoModeWarningRunning { ExternalAccessible := 'False'; ExternalVisible := 'False'; ExternalWritable := 'False'} : DInt;   // Auto Mode warning timmer running / Auto mode warning timmer running
      StartAutoWarning { ExternalAccessible := 'False'; ExternalVisible := 'False'; ExternalWritable := 'False'} : Bool;   // Start button Auto warning
      StartPBSel { ExternalAccessible := 'False'; ExternalVisible := 'False'; ExternalWritable := 'False'} : Bool;   // Summary of Start buttons
      AlarmResetPBSel { ExternalAccessible := 'False'; ExternalVisible := 'False'; ExternalWritable := 'False'} : Bool;   // Summary of Alarm reset buttons
   END_VAR
   VAR
      TimerAutoWarning { ExternalAccessible := 'False'; ExternalVisible := 'False'; ExternalWritable := 'False'} : "LTimer";   // Timer
      TimerResetSequence { ExternalAccessible := 'False'; ExternalVisible := 'False'; ExternalWritable := 'False'} : "LTimer";   // Timer
      TimerAutoNotStarted { ExternalAccessible := 'False'; ExternalVisible := 'False'; ExternalWritable := 'False'} : "LTimer";   // Timer
      TimerStartBtnStuck { ExternalAccessible := 'False'; ExternalVisible := 'False'; ExternalWritable := 'False'} : "LTimer";   // Timer to maximize the pulse on the Start PB
      TimerResetBtnStuck { ExternalAccessible := 'False'; ExternalVisible := 'False'; ExternalWritable := 'False'} : "LTimer";   // Timer to maximize the pulse on the Reset PB
      TimerResetTransportMem { ExternalAccessible := 'False'; ExternalVisible := 'False'; ExternalWritable := 'False'} : "LTimer";   // Timer to extend Reset TM
   END_VAR
   VAR DB_SPECIFIC
      TimerStartPBSel { ExternalAccessible := 'False'; ExternalVisible := 'False'; ExternalWritable := 'False'} : TOF_TIME;   // Timer
      TimerAlarmResetPBSel { ExternalAccessible := 'False'; ExternalVisible := 'False'; ExternalWritable := 'False'} : TOF_TIME;   // Timer
      TimerModeChanged { ExternalAccessible := 'False'; ExternalVisible := 'False'; ExternalWritable := 'False'} : TON_TIME;   // Timer
      TimerScreenChanged { ExternalAccessible := 'False'; ExternalVisible := 'False'; ExternalWritable := 'False'} : TON_TIME;   // Timer
   END_VAR
   VAR_TEMP
      AutoModeWarnMillieSec : DInt;   // Auto Mode warning millie seconds / Auto mode warning millie seconds
      AutoModeWarnSec : DInt;   // Auto Mode warning seconds / Auto mode warning seconds
      AlarmABConditionActive : Bool;   // Alarm AB condition Active in the Modezone / Alarm AB condition
      AlarmAActive : Bool;   // Alarm A Active in the Modezone
      AlarmBActive : Bool;   // Alarm B Active in the Modezone
      AlarmCActive : Bool;   // Alarm C Active in the Modezone
      AlarmDActive : Bool;   // Alarm D Active in the Modezone
   END_VAR
   VAR_TEMP   // added for the SCL form of the ladder/FBD networks
      _w1 : Bool;
      _w2 : Bool;
   END_VAR
BEGIN

REGION Network 1: **** 1 - Inputs **** The Mode has changed
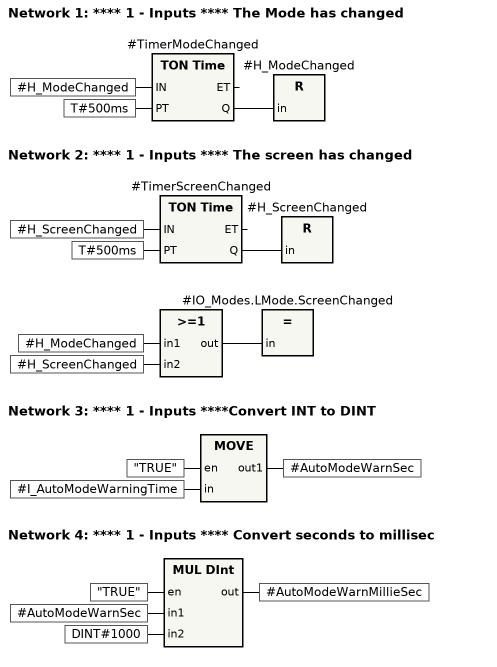
   #TimerModeChanged(IN := #H_ModeChanged, PT := T#500ms);   // TON
   IF #TimerModeChanged.Q THEN #H_ModeChanged := FALSE; END_IF;
END_REGION

REGION Network 2: **** 1 - Inputs **** The screen has changed
   #TimerScreenChanged(IN := #H_ScreenChanged, PT := T#500ms);   // TON
   IF #TimerScreenChanged.Q THEN #H_ScreenChanged := FALSE; END_IF;
   #IO_Modes.LMode.ScreenChanged := #H_ModeChanged OR #H_ScreenChanged;
END_REGION

REGION Network 3: **** 1 - Inputs ****Convert INT to DINT
   // Convert INT to DINT
   IF "TRUE" THEN #AutoModeWarnSec := #I_AutoModeWarningTime; END_IF;
END_REGION

REGION Network 4: **** 1 - Inputs **** Convert seconds to millisec
   // Convert seconds to millisec
   IF "TRUE" THEN #AutoModeWarnMillieSec := #AutoModeWarnSec * DINT#1000; END_IF;
END_REGION

REGION Network 5: **** 1 - Inputs **** Alarms Upperlevel And ModeZone Objects
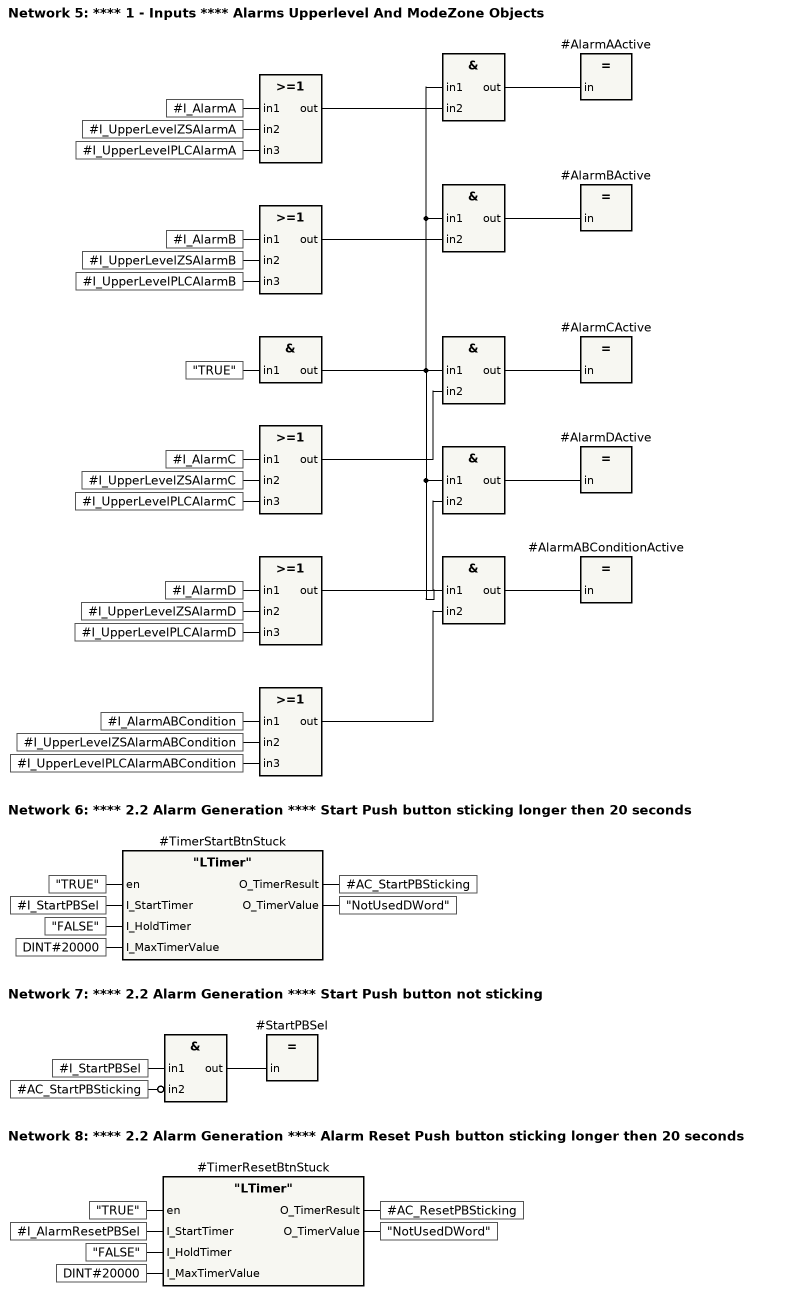
   #AlarmAActive := "TRUE" AND (#I_AlarmA OR #I_UpperLevelZSAlarmA OR #I_UpperLevelPLCAlarmA);
   #AlarmBActive := "TRUE" AND (#I_AlarmB OR #I_UpperLevelZSAlarmB OR #I_UpperLevelPLCAlarmB);
   #AlarmCActive := "TRUE" AND (#I_AlarmC OR #I_UpperLevelZSAlarmC OR #I_UpperLevelPLCAlarmC);
   #AlarmDActive := "TRUE" AND (#I_AlarmD OR #I_UpperLevelZSAlarmD OR #I_UpperLevelPLCAlarmD);
   #AlarmABConditionActive := "TRUE" AND (#I_AlarmABCondition OR #I_UpperLevelZSAlarmABCondition OR #I_UpperLevelPLCAlarmABCondition);
END_REGION

REGION Network 6: **** 2.2 Alarm Generation **** Start Push button sticking longer then 20 seconds
   // Start Push button sticking longer then 20 seconds
   IF "TRUE" THEN
       #TimerStartBtnStuck(I_StartTimer := #I_StartPBSel,   // "LTimer"
                           I_HoldTimer := "FALSE",
                           I_MaxTimerValue := DINT#20000,
                           O_TimerResult => #AC_StartPBSticking,
                           O_TimerValue => "NotUsedDWord");
   END_IF;
END_REGION

REGION Network 7: **** 2.2 Alarm Generation **** Start Push button not sticking
   // Start Push button not sticking
   #StartPBSel := #I_StartPBSel AND NOT #AC_StartPBSticking;
END_REGION

REGION Network 8: **** 2.2 Alarm Generation **** Alarm Reset Push button sticking longer then 20 seconds
   // Alarm Reset Push button sticking longer then 20 seconds
   IF "TRUE" THEN
       #TimerResetBtnStuck(I_StartTimer := #I_AlarmResetPBSel,   // "LTimer"
                           I_HoldTimer := "FALSE",
                           I_MaxTimerValue := DINT#20000,
                           O_TimerResult => #AC_ResetPBSticking,
                           O_TimerValue => "NotUsedDWord");
   END_IF;
END_REGION

REGION Network 9: **** 2.2 Alarm Generation **** Alarm Reset Push button not sticking
   // Alarm Reset Push button not sticking
